LIN {X 0,Y 517.582,Z 524.387,A -85,B 0,C 180,E1 -5009.502,E2 -5009.502} C_VEL
LIN {X 0,Y 517.228,Z 535.267,A -85,B 0,C 180,E1 -5010.714,E2 -5010.714} C_VEL
LIN {X 0,Y 516.853,Z 543.976,A -85,B 0,C 180,E1 -5011.889,E2 -5011.889} C_VEL
LIN {X 0,Y 516.66,Z 551.467,A -85,B 0,C 180,E1 -5013.109,E2 -5013.109} C_VEL
LIN {X 0,Y 516.519,Z 557.024,A -85,B 0,C 180,E1 -5014.189,E2 -5014.189} C_VEL
LIN {X 0,Y 516.363,Z 563.536,A -85,B 0,C 180,E1 -5015.768,E2 -5015.768} C_VEL
LIN {X 0,Y 516.294,Z 567.941,A -85,B 0,C 180,E1 -5017.173,E2 -5017.173} C_VEL
LIN {X 0,Y 516.226,Z 570.925,A -85,B 0,C 180,E1 -5018.433,E2 -5018.433} C_VEL
LIN {X 0,Y 516.199,Z 573.444,A -85,B 0,C 180,E1 -5020.1,E2 -5020.1} C_VEL
LIN {X 0,Y 516.154,Z 574.446,A -85,B 0,C 180,E1 -5021.749,E2 -5021.749} C_VEL
LIN {X 0,Y 516.194,Z 574.398,A -85,B 0,C 180,E1 -5022.57,E2 -5022.57} C_VEL
LIN {X 0,Y 516.141,Z 573.229,A -85,B 0,C 180,E1 -5024.197,E2 -5024.197} C_VEL
LIN {X 0,Y 516.214,Z 570.618,A -85,B 0,C 180,E1 -5025.814,E2 -5025.814} C_VEL
LIN {X 0,Y 516.335,Z 566.52,A -85,B 0,C 180,E1 -5027.421,E2 -5027.421} C_VEL
LIN {X 0,Y 516.436,Z 560.9,A -85,B 0,C 180,E1 -5029.017,E2 -5029.017} C_VEL
LIN {X 0,Y 516.594,Z 554.564,A -85,B 0,C 180,E1 -5030.406,E2 -5030.406} C_VEL
LIN {X 0,Y 516.803,Z 546.711,A -85,B 0,C 180,E1 -5031.791,E2 -5031.791} C_VEL
LIN {X 0,Y 517.103,Z 538.503,A -85,B 0,C 180,E1 -5032.974,E2 -5032.974} C_VEL
LIN {X 0,Y 517.456,Z 528.649,A -85,B 0,C 180,E1 -5034.153,E2 -5034.153} C_VEL
LIN {X 0,Y 517.845,Z 517.719,A -85,B 0,C 180,E1 -5035.232,E2 -5035.232} C_VEL
LIN {X 0,Y 518.215,Z 506.878,A -85,B 0,C 180,E1 -5036.112,E2 -5036.112} C_VEL
LIN {X 0,Y 518.592,Z 495.168,A -85,B 0,C 180,E1 -5036.892,E2 -5036.892} C_VEL
LIN {X 0,Y 518.99,Z 482.323,A -85,B 0,C 180,E1 -5037.574,E2 -5037.574} C_VEL
LIN {X 0,Y 519.323,Z 468.411,A -85,B 0,C 180,E1 -5038.134,E2 -5038.134} C_VEL
LIN {X 0,Y 519.295,Z 460.742,A -85,B 0,C 180,E1 -5038.376,E2 -5038.376} C_VEL
LIN {X 0,Y 516.314,Z 447.75,A -85,B 0,C 180,E1 -5038.781,E2 -5038.781} C_VEL
LIN {X 0,Y 516.336,Z 445.185,A -85,B 0,C 180,E1 -5041.56,E2 -5041.56} C_VEL
LIN {X 0,Y 516.516,Z 443.11,A -85,B 0,C 180,E1 -5043.901,E2 -5043.901} C_VEL
LIN {X 0,Y 516.559,Z 440.324,A -85,B 0,C 180,E1 -5047.033,E2 -5047.033} C_VEL
LIN {X 0,Y 516.578,Z 438.281,A -85,B 0,C 180,E1 -5049.396,E2 -5049.396} C_VEL
LIN {X 0,Y 516.651,Z 436.223,A -85,B 0,C 180,E1 -5051.773,E2 -5051.773} C_VEL
LIN {X 0,Y 516.721,Z 433.411,A -85,B 0,C 180,E1 -5055.058,E2 -5055.058} C_VEL
LIN {X 0,Y 516.78,Z 430.702,A -85,B 0,C 180,E1 -5058.227,E2 -5058.227} C_VEL
LIN {X 0,Y 516.821,Z 429.737,A -85,B 0,C 180,E1 -5059.875,E2 -5059.875} C_VEL
LIN {X 0,Y 516.877,Z 429.729,A -85,B 0,C 180,E1 -5062.395,E2 -5062.395} C_VEL
LIN {X 0,Y 516.906,Z 429.721,A -85,B 0,C 180,E1 -5064.928,E2 -5064.928} C_VEL
LIN {X 0,Y 516.922,Z 429.723,A -85,B 0,C 180,E1 -5067.906,E2 -5067.906} C_VEL
LIN {X 0,Y 516.897,Z 429.726,A -85,B 0,C 180,E1 -5070.203,E2 -5070.203} C_VEL
LIN {X 0,Y 516.893,Z 429.722,A -85,B 0,C 180,E1 -5072.947,E2 -5072.947} C_VEL
LIN {X 0,Y 516.886,Z 429.728,A -85,B 0,C 180,E1 -5075.779,E2 -5075.779} C_VEL
LIN {X 0,Y 516.882,Z 429.724,A -85,B 0,C 180,E1 -5078.716,E2 -5078.716} C_VEL
LIN {X 0,Y 516.915,Z 429.724,A -85,B 0,C 180,E1 -5081.775,E2 -5081.775} C_VEL
LIN {X 0,Y 516.919,Z 429.724,A -85,B 0,C 180,E1 -5085.011,E2 -5085.011} C_VEL
LIN {X 0,Y 516.903,Z 429.871,A -85,B 0,C 180,E1 -5087.039,E2 -5087.039} C_VEL
LIN {X 0,Y 517.709,Z 434.112,A -85,B 0,C 180,E1 -5089.483,E2 -5089.483} C_VEL
LIN {X 0,Y 518.164,Z 437.995,A -85,B 0,C 180,E1 -5091.399,E2 -5091.399} C_VEL
LIN {X 0,Y 517.907,Z 443.605,A -85,B 0,C 180,E1 -5093.823,E2 -5093.823} C_VEL
LIN {X 0,Y 517.585,Z 450.744,A -85,B 0,C 180,E1 -5096.639,E2 -5096.639} C_VEL
LIN {X 0,Y 517.384,Z 456.944,A -85,B 0,C 180,E1 -5098.924,E2 -5098.924} C_VEL
LIN {X 0,Y 517.204,Z 465.92,A -85,B 0,C 180,E1 -5102.037,E2 -5102.037} C_VEL
LIN {X 0,Y 517.018,Z 473.813,A -85,B 0,C 180,E1 -5104.648,E2 -5104.648} C_VEL
LIN {X 0,Y 516.875,Z 483.182,A -85,B 0,C 180,E1 -5107.622,E2 -5107.622} C_VEL
LIN {X 0,Y 516.76,Z 492.685,A -85,B 0,C 180,E1 -5110.537,E2 -5110.537} C_VEL
LIN {X 0,Y 516.657,Z 501.369,A -85,B 0,C 180,E1 -5113.199,E2 -5113.199} C_VEL
LIN {X 0,Y 519.498,Z 516.364,A -85,B 0,C 180,E1 -5113.597,E2 -5113.597} C_VEL
LIN {X 0,Y 519.215,Z 529.798,A -85,B 0,C 180,E1 -5114.012,E2 -5114.012} C_VEL
LIN {X 0,Y 518.816,Z 543.3,A -85,B 0,C 180,E1 -5114.583,E2 -5114.583} C_VEL
LIN {X 0,Y 518.474,Z 555.946,A -85,B 0,C 180,E1 -5115.277,E2 -5115.277} C_VEL
LIN {X 0,Y 518.033,Z 568.91,A -85,B 0,C 180,E1 -5116.166,E2 -5116.166} C_VEL
LIN {X 0,Y 517.648,Z 580.606,A -85,B 0,C 180,E1 -5117.155,E2 -5117.155} C_VEL
LIN {X 0,Y 517.328,Z 591.208,A -85,B 0,C 180,E1 -5118.242,E2 -5118.242} C_VEL
LIN {X 0,Y 517.002,Z 600.782,A -85,B 0,C 180,E1 -5119.426,E2 -5119.426} C_VEL
LIN {X 0,Y 516.77,Z 608.636,A -85,B 0,C 180,E1 -5120.608,E2 -5120.608} C_VEL
LIN {X 0,Y 516.576,Z 615.134,A -85,B 0,C 180,E1 -5121.787,E2 -5121.787} C_VEL
LIN {X 0,Y 516.406,Z 620.528,A -85,B 0,C 180,E1 -5122.965,E2 -5122.965} C_VEL
LIN {X 0,Y 516.407,Z 624.961,A -85,B 0,C 180,E1 -5124.142,E2 -5124.142} C_VEL
LIN {X 0,Y 516.264,Z 628.444,A -85,B 0,C 180,E1 -5125.315,E2 -5125.315} C_VEL
LIN {X 0,Y 516.276,Z 631.832,A -85,B 0,C 180,E1 -5126.879,E2 -5126.879} C_VEL
LIN {X 0,Y 516.188,Z 633.835,A -85,B 0,C 180,E1 -5128.44,E2 -5128.44} C_VEL
LIN {X 0,Y 516.152,Z 634.5,A -85,B 0,C 180,E1 -5130,E2 -5130} C_VEL
LIN {X 0,Y 516.188,Z 633.837,A -85,B 0,C 180,E1 -5131.56,E2 -5131.56} C_VEL
LIN {X 0,Y 516.276,Z 631.836,A -85,B 0,C 180,E1 -5133.121,E2 -5133.121} C_VEL
LIN {X 0,Y 516.325,Z 630.32,A -85,B 0,C 180,E1 -5133.902,E2 -5133.902} C_VEL
LIN {X 0,Y 516.388,Z 626.201,A -85,B 0,C 180,E1 -5135.467,E2 -5135.467} C_VEL
LIN {X 0,Y 516.406,Z 620.526,A -85,B 0,C 180,E1 -5137.035,E2 -5137.035} C_VEL
LIN {X 0,Y 516.599,Z 614.127,A -85,B 0,C 180,E1 -5138.409,E2 -5138.409} C_VEL
LIN {X 0,Y 516.826,Z 606.174,A -85,B 0,C 180,E1 -5139.786,E2 -5139.786} C_VEL
LIN {X 0,Y 517.109,Z 597.777,A -85,B 0,C 180,E1 -5140.969,E2 -5140.969} C_VEL
LIN {X 0,Y 517.439,Z 587.23,A -85,B 0,C 180,E1 -5142.197,E2 -5142.197} C_VEL
LIN {X 0,Y 517.815,Z 576.321,A -85,B 0,C 180,E1 -5143.24,E2 -5143.24} C_VEL
LIN {X 0,Y 518.231,Z 563.637,A -85,B 0,C 180,E1 -5144.229,E2 -5144.229} C_VEL
LIN {X 0,Y 518.694,Z 551.059,A -85,B 0,C 180,E1 -5145.018,E2 -5145.018} C_VEL
LIN {X 0,Y 519.021,Z 538.132,A -85,B 0,C 180,E1 -5145.662,E2 -5145.662} C_VEL
LIN {X 0,Y 519.346,Z 524.193,A -85,B 0,C 180,E1 -5146.186,E2 -5146.186} C_VEL
LIN {X 0,Y 519.351,Z 515.338,A -85,B 0,C 180,E1 -5146.444,E2 -5146.444} C_VEL
LIN {X 0,Y 516.657,Z 501.675,A -85,B 0,C 180,E1 -5146.801,E2 -5146.801} C_VEL
LIN {X 0,Y 516.81,Z 491.833,A -85,B 0,C 180,E1 -5149.875,E2 -5149.875} C_VEL
LIN {X 0,Y 516.966,Z 482.641,A -85,B 0,C 180,E1 -5152.795,E2 -5152.795} C_VEL
LIN {X 0,Y 517.164,Z 473.559,A -85,B 0,C 180,E1 -5155.776,E2 -5155.776} C_VEL
LIN {X 0,Y 517.398,Z 464.561,A -85,B 0,C 180,E1 -5158.829,E2 -5158.829} C_VEL
LIN {X 0,Y 517.651,Z 456.874,A -85,B 0,C 180,E1 -5161.536,E2 -5161.536} C_VEL
LIN {X 0,Y 517.857,Z 449.76,A -85,B 0,C 180,E1 -5164.121,E2 -5164.121} C_VEL
LIN {X 0,Y 518.122,Z 442.579,A -85,B 0,C 180,E1 -5166.841,E2 -5166.841} C_VEL
LIN {X 0,Y 518.252,Z 438.106,A -85,B 0,C 180,E1 -5168.594,E2 -5168.594} C_VEL
LIN {X 0,Y 517.521,Z 433.141,A -85,B 0,C 180,E1 -5170.68,E2 -5170.68} C_VEL
LIN {X 0,Y 516.901,Z 429.726,A -85,B 0,C 180,E1 -5172.234,E2 -5172.234} C_VEL
LIN {X 0,Y 516.919,Z 429.724,A -85,B 0,C 180,E1 -5175.01,E2 -5175.01} C_VEL
LIN {X 0,Y 516.913,Z 429.72,A -85,B 0,C 180,E1 -5178.398,E2 -5178.398} C_VEL
LIN {X 0,Y 516.878,Z 429.726,A -85,B 0,C 180,E1 -5181.284,E2 -5181.284} C_VEL
LIN {X 0,Y 516.882,Z 429.725,A -85,B 0,C 180,E1 -5184.221,E2 -5184.221} C_VEL
LIN {X 0,Y 516.893,Z 429.725,A -85,B 0,C 180,E1 -5187.053,E2 -5187.053} C_VEL
LIN {X 0,Y 516.897,Z 429.725,A -85,B 0,C 180,E1 -5189.797,E2 -5189.797} C_VEL
LIN {X 0,Y 516.925,Z 429.72,A -85,B 0,C 180,E1 -5192.467,E2 -5192.467} C_VEL
LIN {X 0,Y 516.906,Z 429.723,A -85,B 0,C 180,E1 -5195.072,E2 -5195.072} C_VEL
LIN {X 0,Y 516.881,Z 429.729,A -85,B 0,C 180,E1 -5198.462,E2 -5198.462} C_VEL
LIN {X 0,Y 516.899,Z 429.726,A -85,B 0,C 180,E1 -5200.955,E2 -5200.955} C_VEL
LIN {X 0,Y 516.912,Z 429.722,A -85,B 0,C 180,E1 -5203.41,E2 -5203.41} C_VEL
LIN {X 0,Y 516.888,Z 429.723,A -85,B 0,C 180,E1 -5205.834,E2 -5205.834} C_VEL
LIN {X 0,Y 516.951,Z 429.718,A -85,B 0,C 180,E1 -5209.028,E2 -5209.028} C_VEL
LIN {X 0,Y 516.972,Z 429.717,A -85,B 0,C 180,E1 -5212.187,E2 -5212.187} C_VEL
LIN {X 0,Y 517.026,Z 429.708,A -85,B 0,C 180,E1 -5214.54,E2 -5214.54} C_VEL
LIN {X 0,Y 517.078,Z 429.703,A -85,B 0,C 180,E1 -5217.663,E2 -5217.663} C_VEL
LIN {X 0,Y 517.088,Z 429.7,A -85,B 0,C 180,E1 -5220.779,E2 -5220.779} C_VEL
LIN {X 0,Y 517.011,Z 429.711,A -85,B 0,C 180,E1 -5223.117,E2 -5223.117} C_VEL
LIN {X 0,Y 517.01,Z 429.71,A -85,B 0,C 180,E1 -5226.243,E2 -5226.243} C_VEL
LIN {X 0,Y 516.951,Z 429.716,A -85,B 0,C 180,E1 -5229.389,E2 -5229.389} C_VEL
LIN {X 0,Y 516.945,Z 429.718,A -85,B 0,C 180,E1 -5231.808,E2 -5231.808} C_VEL
LIN {X 0,Y 516.938,Z 429.72,A -85,B 0,C 180,E1 -5235.147,E2 -5235.147} C_VEL
LIN {X 0,Y 516.92,Z 429.724,A -85,B 0,C 180,E1 -5238.223,E2 -5238.223} C_VEL
LIN {X 0,Y 516.908,Z 429.724,A -85,B 0,C 180,E1 -5240.702,E2 -5240.702} C_VEL
LIN {X 0,Y 516.906,Z 429.724,A -85,B 0,C 180,E1 -5244.073,E2 -5244.073} C_VEL
LIN {X 0,Y 516.921,Z 429.721,A -85,B 0,C 180,E1 -5246.658,E2 -5246.658} C_VEL
LIN {X 0,Y 516.907,Z 429.724,A -85,B 0,C 180,E1 -5249.525,E2 -5249.525} C_VEL
LIN {X 0,Y 516.897,Z 429.723,A -85,B 0,C 180,E1 -5252.545,E2 -5252.545} C_VEL
LIN {X 0,Y 516.877,Z 429.725,A -85,B 0,C 180,E1 -5255.333,E2 -5255.333} C_VEL
LIN {X 0,Y 516.878,Z 429.726,A -85,B 0,C 180,E1 -5257.944,E2 -5257.944} C_VEL
LIN {X 0,Y 516.881,Z 429.724,A -85,B 0,C 180,E1 -5260.742,E2 -5260.742} C_VEL
LIN {X 0,Y 516.903,Z 429.725,A -85,B 0,C 180,E1 -5262.83,E2 -5262.83} C_VEL
LIN {X 0,Y 516.921,Z 429.719,A -85,B 0,C 180,E1 -5265.011,E2 -5265.011} C_VEL
LIN {X 0,Y 516.914,Z 429.724,A -85,B 0,C 180,E1 -5268.399,E2 -5268.399} C_VEL
LIN {X 0,Y 516.892,Z 429.724,A -85,B 0,C 180,E1 -5270.313,E2 -5270.313} C_VEL
LIN {X 0,Y 516.22,Z 429.809,A -85,B 0,C 180,E1 -5270.963,E2 -5270.963} C_VEL
LIN {X 0,Y 513.369,Z 430.165,A -85,B 0,C 180,E1 -5272.019,E2 -5272.019} C_VEL
LIN {X 0,Y 510.96,Z 430.466,A -85,B 0,C 180,E1 -5272.869,E2 -5272.869} C_VEL
LIN {X 0,Y 509.92,Z 430.594,A -85,B 0,C 180,E1 -5273.526,E2 -5273.526} C_VEL
LIN {X 0,Y 509.832,Z 430.604,A -85,B 0,C 180,E1 -5273.748,E2 -5273.748} C_VEL
LIN {X 0,Y 509.863,Z 430.602,A -85,B 0,C 180,E1 -5276.54,E2 -5276.54} C_VEL
LIN {X 0,Y 509.851,Z 430.602,A -85,B 0,C 180,E1 -5279.335,E2 -5279.335} C_VEL
LIN {X 0,Y 509.896,Z 430.599,A -85,B 0,C 180,E1 -5282.055,E2 -5282.055} C_VEL
LIN {X 0,Y 509.879,Z 430.599,A -85,B 0,C 180,E1 -5284.705,E2 -5284.705} C_VEL
LIN {X 0,Y 509.829,Z 430.605,A -85,B 0,C 180,E1 -5287.458,E2 -5287.458} C_VEL
LIN {X 0,Y 509.92,Z 430.593,A -85,B 0,C 180,E1 -5289.845,E2 -5289.845} C_VEL
LIN {X 0,Y 509.886,Z 430.599,A -85,B 0,C 180,E1 -5293.175,E2 -5293.175} C_VEL
LIN {X 0,Y 509.868,Z 430.6,A -85,B 0,C 180,E1 -5295.635,E2 -5295.635} C_VEL
LIN {X 0,Y 509.917,Z 430.595,A -85,B 0,C 180,E1 -5298.875,E2 -5298.875} C_VEL
LIN {X 0,Y 509.955,Z 430.588,A -85,B 0,C 180,E1 -5302.079,E2 -5302.079} C_VEL
LIN {X 0,Y 509.979,Z 430.586,A -85,B 0,C 180,E1 -5304.464,E2 -5304.464} C_VEL
LIN {X 0,Y 510.059,Z 430.575,A -85,B 0,C 180,E1 -5307.631,E2 -5307.631} C_VEL
LIN {X 0,Y 510.067,Z 430.574,A -85,B 0,C 180,E1 -5310.789,E2 -5310.789} C_VEL
LIN {X 0,Y 509.958,Z 430.588,A -85,B 0,C 180,E1 -5313.16,E2 -5313.16} C_VEL
LIN {X 0,Y 509.984,Z 430.586,A -85,B 0,C 180,E1 -5316.329,E2 -5316.329} C_VEL
LIN {X 0,Y 509.895,Z 430.597,A -85,B 0,C 180,E1 -5319.52,E2 -5319.52} C_VEL
LIN {X 0,Y 509.909,Z 430.596,A -85,B 0,C 180,E1 -5321.931,E2 -5321.931} C_VEL
LIN {X 0,Y 509.898,Z 430.596,A -85,B 0,C 180,E1 -5325.241,E2 -5325.241} C_VEL
LIN {X 0,Y 509.885,Z 430.596,A -85,B 0,C 180,E1 -5327.998,E2 -5327.998} C_VEL
LIN {X 0,Y 509.853,Z 430.601,A -85,B 0,C 180,E1 -5331.001,E2 -5331.001} C_VEL
LIN {X 0,Y 509.873,Z 430.6,A -85,B 0,C 180,E1 -5334.425,E2 -5334.425} C_VEL
LIN {X 0,Y 509.888,Z 430.599,A -85,B 0,C 180,E1 -5337.055,E2 -5337.055} C_VEL
LIN {X 0,Y 509.859,Z 430.602,A -85,B 0,C 180,E1 -5339.75,E2 -5339.75} C_VEL
LIN {X 0,Y 509.846,Z 430.605,A -85,B 0,C 180,E1 -5342.769,E2 -5342.769} C_VEL
LIN {X 0,Y 509.695,Z 430.624,A -85,B 0,C 180,E1 -5345.557,E2 -5345.557} C_VEL
LIN {X 0,Y 509.451,Z 430.654,A -85,B 0,C 180,E1 -5347.371,E2 -5347.371} C_VEL
LIN {X 0,Y 509.404,Z 432.343,A -85,B 0,C 180,E1 -5349.411,E2 -5349.411} C_VEL
LIN {X 0,Y 509.366,Z 435.356,A -85,B 0,C 180,E1 -5352.537,E2 -5352.537} C_VEL
LIN {X 0,Y 509.316,Z 438.013,A -85,B 0,C 180,E1 -5355.271,E2 -5355.271} C_VEL
LIN {X 0,Y 509.301,Z 440.829,A -85,B 0,C 180,E1 -5358.172,E2 -5358.172} C_VEL
LIN {X 0,Y 509.23,Z 443.23,A -85,B 0,C 180,E1 -5360.611,E2 -5360.611} C_VEL
LIN {X 0,Y 509.173,Z 446.185,A -85,B 0,C 180,E1 -5363.593,E2 -5363.593} C_VEL
LIN {X 0,Y 509.185,Z 447.643,A -85,B 0,C 180,E1 -5365.053,E2 -5365.053} C_VEL
LIN {X 0,Y 512.553,Z 462.05,A -85,B 0,C 180,E1 -5365.528,E2 -5365.528} C_VEL
LIN {X 0,Y 512.339,Z 475.814,A -85,B 0,C 180,E1 -5366.014,E2 -5366.014} C_VEL
LIN {X 0,Y 511.944,Z 488.952,A -85,B 0,C 180,E1 -5366.634,E2 -5366.634} C_VEL
LIN {X 0,Y 511.538,Z 501.39,A -85,B 0,C 180,E1 -5367.387,E2 -5367.387} C_VEL
LIN {X 0,Y 511.091,Z 513.106,A -85,B 0,C 180,E1 -5368.266,E2 -5368.266} C_VEL
LIN {X 0,Y 510.661,Z 524.126,A -85,B 0,C 180,E1 -5369.274,E2 -5369.274} C_VEL
LIN {X 0,Y 510.337,Z 533.322,A -85,B 0,C 180,E1 -5370.279,E2 -5370.279} C_VEL
LIN {X 0,Y 509.919,Z 543.164,A -85,B 0,C 180,E1 -5371.58,E2 -5371.58} C_VEL
LIN {X 0,Y 509.658,Z 551.503,A -85,B 0,C 180,E1 -5372.931,E2 -5372.931} C_VEL
LIN {X 0,Y 509.447,Z 558.111,A -85,B 0,C 180,E1 -5374.243,E2 -5374.243} C_VEL
LIN {X 0,Y 509.33,Z 563.618,A -85,B 0,C 180,E1 -5375.6,E2 -5375.6} C_VEL
LIN {X 0,Y 509.23,Z 567.618,A -85,B 0,C 180,E1 -5376.838,E2 -5376.838} C_VEL
LIN {X 0,Y 509.176,Z 570.752,A -85,B 0,C 180,E1 -5378.119,E2 -5378.119} C_VEL
LIN {X 0,Y 509.132,Z 572.341,A -85,B 0,C 180,E1 -5378.967,E2 -5378.967} C_VEL
LIN {X 0,Y 509.092,Z 574.299,A -85,B 0,C 180,E1 -5380.651,E2 -5380.651} C_VEL
LIN {X 0,Y 509.099,Z 574.776,A -85,B 0,C 180,E1 -5382.319,E2 -5382.319} C_VEL
LIN {X 0,Y 509.047,Z 573.836,A -85,B 0,C 180,E1 -5383.971,E2 -5383.971} C_VEL
LIN {X 0,Y 509.118,Z 571.48,A -85,B 0,C 180,E1 -5385.612,E2 -5385.612} C_VEL
LIN {X 0,Y 509.258,Z 567.68,A -85,B 0,C 180,E1 -5387.243,E2 -5387.243} C_VEL
LIN {X 0,Y 509.312,Z 563.858,A -85,B 0,C 180,E1 -5388.439,E2 -5388.439} C_VEL
LIN {X 0,Y 509.45,Z 558.988,A -85,B 0,C 180,E1 -5389.669,E2 -5389.669} C_VEL
LIN {X 0,Y 509.633,Z 552.069,A -85,B 0,C 180,E1 -5391.075,E2 -5391.075} C_VEL
LIN {X 0,Y 509.959,Z 543.497,A -85,B 0,C 180,E1 -5392.477,E2 -5392.477} C_VEL
LIN {X 0,Y 510.297,Z 534.568,A -85,B 0,C 180,E1 -5393.674,E2 -5393.674} C_VEL
LIN {X 0,Y 510.667,Z 523.806,A -85,B 0,C 180,E1 -5394.868,E2 -5394.868} C_VEL
LIN {X 0,Y 511.069,Z 512.891,A -85,B 0,C 180,E1 -5395.86,E2 -5395.86} C_VEL
LIN {X 0,Y 511.544,Z 500.871,A -85,B 0,C 180,E1 -5396.751,E2 -5396.751} C_VEL
LIN {X 0,Y 511.949,Z 489.396,A -85,B 0,C 180,E1 -5397.443,E2 -5397.443} C_VEL
LIN {X 0,Y 512.396,Z 475.758,A -85,B 0,C 180,E1 -5398.084,E2 -5398.084} C_VEL
LIN {X 0,Y 512.533,Z 462.151,A -85,B 0,C 180,E1 -5398.563,E2 -5398.563} C_VEL
LIN {X 0,Y 509.833,Z 450.501,A -85,B 0,C 180,E1 -5398.951,E2 -5398.951} C_VEL
LIN {X 0,Y 509.262,Z 448.284,A -85,B 0,C 180,E1 -5399.011,E2 -5399.011} C_VEL
LIN {X 0,Y 509.279,Z 445.95,A -85,B 0,C 180,E1 -5401.581,E2 -5401.581} C_VEL
LIN {X 0,Y 509.47,Z 443.813,A -85,B 0,C 180,E1 -5403.955,E2 -5403.955} C_VEL
LIN {X 0,Y 509.518,Z 441.038,A -85,B 0,C 180,E1 -5407.131,E2 -5407.131} C_VEL
LIN {X 0,Y 509.524,Z 438.956,A -85,B 0,C 180,E1 -5409.527,E2 -5409.527} C_VEL
LIN {X 0,Y 509.606,Z 436.898,A -85,B 0,C 180,E1 -5411.939,E2 -5411.939} C_VEL
LIN {X 0,Y 509.68,Z 434.149,A -85,B 0,C 180,E1 -5415.188,E2 -5415.188} C_VEL
LIN {X 0,Y 509.756,Z 431.418,A -85,B 0,C 180,E1 -5418.488,E2 -5418.488} C_VEL
LIN {X 0,Y 509.761,Z 430.758,A -85,B 0,C 180,E1 -5419.322,E2 -5419.322} C_VEL
LIN {X 0,Y 509.807,Z 430.61,A -85,B 0,C 180,E1 -5421.852,E2 -5421.852} C_VEL
LIN {X 0,Y 509.854,Z 430.603,A -85,B 0,C 180,E1 -5424.529,E2 -5424.529} C_VEL
LIN {X 0,Y 509.882,Z 430.596,A -85,B 0,C 180,E1 -5427.056,E2 -5427.056} C_VEL
LIN {X 0,Y 509.875,Z 430.599,A -85,B 0,C 180,E1 -5429.75,E2 -5429.75} C_VEL
LIN {X 0,Y 509.872,Z 430.597,A -85,B 0,C 180,E1 -5432.775,E2 -5432.775} C_VEL
LIN {X 0,Y 509.838,Z 430.604,A -85,B 0,C 180,E1 -5435.582,E2 -5435.582} C_VEL
LIN {X 0,Y 509.847,Z 430.603,A -85,B 0,C 180,E1 -5438.338,E2 -5438.338} C_VEL
LIN {X 0,Y 509.862,Z 430.601,A -85,B 0,C 180,E1 -5441.425,E2 -5441.425} C_VEL
LIN {X 0,Y 509.853,Z 430.605,A -85,B 0,C 180,E1 -5444.668,E2 -5444.668} C_VEL
LIN {X 0,Y 509.864,Z 430.81,A -85,B 0,C 180,E1 -5446.647,E2 -5446.647} C_VEL
LIN {X 0,Y 510.85,Z 436.046,A -85,B 0,C 180,E1 -5449.715,E2 -5449.715} C_VEL
LIN {X 0,Y 511.211,Z 440.221,A -85,B 0,C 180,E1 -5451.783,E2 -5451.783} C_VEL
LIN {X 0,Y 510.839,Z 447.028,A -85,B 0,C 180,E1 -5454.703,E2 -5454.703} C_VEL
LIN {X 0,Y 510.496,Z 454.238,A -85,B 0,C 180,E1 -5457.527,E2 -5457.527} C_VEL
LIN {X 0,Y 510.327,Z 460.494,A -85,B 0,C 180,E1 -5459.823,E2 -5459.823} C_VEL
LIN {X 0,Y 510.071,Z 469.506,A -85,B 0,C 180,E1 -5462.956,E2 -5462.956} C_VEL
LIN {X 0,Y 509.877,Z 478.717,A -85,B 0,C 180,E1 -5466.008,E2 -5466.008} C_VEL
LIN {X 0,Y 509.742,Z 486.765,A -85,B 0,C 180,E1 -5468.57,E2 -5468.57} C_VEL
LIN {X 0,Y 509.638,Z 496.174,A -85,B 0,C 180,E1 -5471.508,E2 -5471.508} C_VEL
LIN {X 0,Y 509.567,Z 500.902,A -85,B 0,C 180,E1 -5472.968,E2 -5472.968} C_VEL
LIN {X 0,Y 511.963,Z 513.726,A -85,B 0,C 180,E1 -5473.302,E2 -5473.302} C_VEL
LIN {X 0,Y 512.586,Z 518.364,A -85,B 0,C 180,E1 -5473.446,E2 -5473.446} C_VEL
LIN {X 0,Y 512.279,Z 532.267,A -85,B 0,C 180,E1 -5473.914,E2 -5473.914} C_VEL
LIN {X 0,Y 511.88,Z 544.613,A -85,B 0,C 180,E1 -5474.471,E2 -5474.471} C_VEL
LIN {X 0,Y 511.453,Z 558.471,A -85,B 0,C 180,E1 -5475.273,E2 -5475.273} C_VEL
LIN {X 0,Y 510.973,Z 570.86,A -85,B 0,C 180,E1 -5476.174,E2 -5476.174} C_VEL
LIN {X 0,Y 510.562,Z 582.106,A -85,B 0,C 180,E1 -5477.176,E2 -5477.176} C_VEL
LIN {X 0,Y 510.255,Z 592.36,A -85,B 0,C 180,E1 -5478.278,E2 -5478.278} C_VEL
LIN {X 0,Y 509.889,Z 601.645,A -85,B 0,C 180,E1 -5479.477,E2 -5479.477} C_VEL
LIN {X 0,Y 509.604,Z 610.518,A -85,B 0,C 180,E1 -5480.875,E2 -5480.875} C_VEL
LIN {X 0,Y 509.424,Z 616.768,A -85,B 0,C 180,E1 -5482.07,E2 -5482.07} C_VEL
LIN {X 0,Y 509.308,Z 623.403,A -85,B 0,C 180,E1 -5483.662,E2 -5483.662} C_VEL
LIN {X 0,Y 509.239,Z 627.283,A -85,B 0,C 180,E1 -5484.853,E2 -5484.853} C_VEL
LIN {X 0,Y 509.218,Z 630.271,A -85,B 0,C 180,E1 -5486.043,E2 -5486.043} C_VEL
LIN {X 0,Y 509.159,Z 632.991,A -85,B 0,C 180,E1 -5487.627,E2 -5487.627} C_VEL
LIN {X 0,Y 509.071,Z 634.33,A -85,B 0,C 180,E1 -5489.209,E2 -5489.209} C_VEL
LIN {X 0,Y 509.071,Z 634.33,A -85,B 0,C 180,E1 -5490.791,E2 -5490.791} C_VEL
LIN {X 0,Y 509.159,Z 632.994,A -85,B 0,C 180,E1 -5492.373,E2 -5492.373} C_VEL
LIN {X 0,Y 509.218,Z 630.276,A -85,B 0,C 180,E1 -5493.957,E2 -5493.957} C_VEL
LIN {X 0,Y 509.301,Z 626.092,A -85,B 0,C 180,E1 -5495.543,E2 -5495.543} C_VEL
LIN {X 0,Y 509.329,Z 620.324,A -85,B 0,C 180,E1 -5497.134,E2 -5497.134} C_VEL
LIN {X 0,Y 509.535,Z 613.831,A -85,B 0,C 180,E1 -5498.527,E2 -5498.527} C_VEL
LIN {X 0,Y 509.762,Z 605.761,A -85,B 0,C 180,E1 -5499.923,E2 -5499.923} C_VEL
LIN {X 0,Y 510.066,Z 597.324,A -85,B 0,C 180,E1 -5501.122,E2 -5501.122} C_VEL
LIN {X 0,Y 510.41,Z 587.128,A -85,B 0,C 180,E1 -5502.328,E2 -5502.328} C_VEL
LIN {X 0,Y 510.839,Z 575.836,A -85,B 0,C 180,E1 -5503.424,E2 -5503.424} C_VEL
LIN {X 0,Y 511.27,Z 563.136,A -85,B 0,C 180,E1 -5504.427,E2 -5504.427} C_VEL
LIN {X 0,Y 511.772,Z 550.544,A -85,B 0,C 180,E1 -5505.226,E2 -5505.226} C_VEL
LIN {X 0,Y 512.165,Z 537.602,A -85,B 0,C 180,E1 -5505.877,E2 -5505.877} C_VEL
LIN {X 0,Y 512.472,Z 523.802,A -85,B 0,C 180,E1 -5506.404,E2 -5506.404} C_VEL
LIN {X 0,Y 512.475,Z 516.194,A -85,B 0,C 180,E1 -5506.632,E2 -5506.632} C_VEL
LIN {X 0,Y 509.592,Z 501.309,A -85,B 0,C 180,E1 -5507.041,E2 -5507.041} C_VEL
LIN {X 0,Y 509.755,Z 491.493,A -85,B 0,C 180,E1 -5510.162,E2 -5510.162} C_VEL
LIN {X 0,Y 509.935,Z 482.371,A -85,B 0,C 180,E1 -5513.128,E2 -5513.128} C_VEL
LIN {X 0,Y 510.16,Z 473.342,A -85,B 0,C 180,E1 -5516.157,E2 -5516.157} C_VEL
LIN {X 0,Y 510.389,Z 464.396,A -85,B 0,C 180,E1 -5519.263,E2 -5519.263} C_VEL
LIN {X 0,Y 510.65,Z 456.782,A -85,B 0,C 180,E1 -5521.996,E2 -5521.996} C_VEL
LIN {X 0,Y 510.933,Z 449.238,A -85,B 0,C 180,E1 -5524.808,E2 -5524.808} C_VEL
LIN {X 0,Y 511.246,Z 441.72,A -85,B 0,C 180,E1 -5527.714,E2 -5527.714} C_VEL
LIN {X 0,Y 511.137,Z 437.999,A -85,B 0,C 180,E1 -5529.233,E2 -5529.233} C_VEL
LIN {X 0,Y 510.079,Z 431.818,A -85,B 0,C 180,E1 -5531.925,E2 -5531.925} C_VEL
LIN {X 0,Y 509.871,Z 430.601,A -85,B 0,C 180,E1 -5532.485,E2 -5532.485} C_VEL
LIN {X 0,Y 509.853,Z 430.603,A -85,B 0,C 180,E1 -5535.332,E2 -5535.332} C_VEL
LIN {X 0,Y 509.854,Z 430.6,A -85,B 0,C 180,E1 -5538.574,E2 -5538.574} C_VEL
LIN {X 0,Y 509.847,Z 430.605,A -85,B 0,C 180,E1 -5541.786,E2 -5541.786} C_VEL
LIN {X 0,Y 509.838,Z 430.605,A -85,B 0,C 180,E1 -5544.623,E2 -5544.623} C_VEL
LIN {X 0,Y 509.861,Z 430.601,A -85,B 0,C 180,E1 -5547.481,E2 -5547.481} C_VEL
LIN {X 0,Y 509.876,Z 430.6,A -85,B 0,C 180,E1 -5550.269,E2 -5550.269} C_VEL
LIN {X 0,Y 509.882,Z 430.6,A -85,B 0,C 180,E1 -5552.944,E2 -5552.944} C_VEL
LIN {X 0,Y 509.864,Z 430.602,A -85,B 0,C 180,E1 -5555.574,E2 -5555.574} C_VEL
LIN {X 0,Y 509.816,Z 430.606,A -85,B 0,C 180,E1 -5558.148,E2 -5558.148} C_VEL
LIN {X 0,Y 509.859,Z 430.601,A -85,B 0,C 180,E1 -5560.681,E2 -5560.681} C_VEL
LIN {X 0,Y 509.881,Z 430.597,A -85,B 0,C 180,E1 -5563.175,E2 -5563.175} C_VEL
LIN {X 0,Y 509.857,Z 430.6,A -85,B 0,C 180,E1 -5565.634,E2 -5565.634} C_VEL
LIN {X 0,Y 509.911,Z 430.594,A -85,B 0,C 180,E1 -5568.875,E2 -5568.875} C_VEL
LIN {X 0,Y 509.945,Z 430.591,A -85,B 0,C 180,E1 -5572.078,E2 -5572.078} C_VEL
LIN {X 0,Y 509.978,Z 430.586,A -85,B 0,C 180,E1 -5574.464,E2 -5574.464} C_VEL
LIN {X 0,Y 510.049,Z 430.578,A -85,B 0,C 180,E1 -5577.631,E2 -5577.631} C_VEL
LIN {X 0,Y 510.058,Z 430.576,A -85,B 0,C 180,E1 -5580.79,E2 -5580.79} C_VEL
LIN {X 0,Y 509.954,Z 430.59,A -85,B 0,C 180,E1 -5583.16,E2 -5583.16} C_VEL
LIN {X 0,Y 509.977,Z 430.586,A -85,B 0,C 180,E1 -5586.33,E2 -5586.33} C_VEL
LIN {X 0,Y 509.912,Z 430.595,A -85,B 0,C 180,E1 -5588.72,E2 -5588.72} C_VEL
LIN {X 0,Y 509.897,Z 430.595,A -85,B 0,C 180,E1 -5591.932,E2 -5591.932} C_VEL
LIN {X 0,Y 509.887,Z 430.598,A -85,B 0,C 180,E1 -5595.242,E2 -5595.242} C_VEL
LIN {X 0,Y 509.883,Z 430.598,A -85,B 0,C 180,E1 -5598.002,E2 -5598.002} C_VEL
LIN {X 0,Y 509.845,Z 430.604,A -85,B 0,C 180,E1 -5601.002,E2 -5601.002} C_VEL
LIN {X 0,Y 509.831,Z 430.605,A -85,B 0,C 180,E1 -5603.564,E2 -5603.564} C_VEL
LIN {X 0,Y 509.907,Z 430.597,A -85,B 0,C 180,E1 -5606.379,E2 -5606.379} C_VEL
LIN {X 0,Y 509.872,Z 430.599,A -85,B 0,C 180,E1 -5608.845,E2 -5608.845} C_VEL
LIN {X 0,Y 509.821,Z 430.604,A -85,B 0,C 180,E1 -5611.59,E2 -5611.59} C_VEL
LIN {X 0,Y 509.849,Z 430.603,A -85,B 0,C 180,E1 -5614.414,E2 -5614.414} C_VEL
LIN {X 0,Y 509.815,Z 430.607,A -85,B 0,C 180,E1 -5617.341,E2 -5617.341} C_VEL
LIN {X 0,Y 509.835,Z 430.604,A -85,B 0,C 180,E1 -5620.383,E2 -5620.383} C_VEL
LIN {X 0,Y 509.838,Z 430.604,A -85,B 0,C 180,E1 -5623.065,E2 -5623.065} C_VEL
LIN {X 0,Y 509.829,Z 430.607,A -85,B 0,C 180,E1 -5625.793,E2 -5625.793} C_VEL
LIN {X 0,Y 509.857,Z 430.602,A -85,B 0,C 180,E1 -5628.576,E2 -5628.576} C_VEL
LIN {X 0,Y 509.852,Z 430.601,A -85,B 0,C 180,E1 -5631.787,E2 -5631.787} C_VEL
LIN {X 0,Y 509.832,Z 430.604,A -85,B 0,C 180,E1 -5633.748,E2 -5633.748} C_VEL
LIN {X 0,Y 509.167,Z 430.686,A -85,B 0,C 180,E1 -5634.408,E2 -5634.408} C_VEL
LIN {X 0,Y 506.349,Z 431.04,A -85,B 0,C 180,E1 -5635.48,E2 -5635.48} C_VEL
LIN {X 0,Y 503.955,Z 431.338,A -85,B 0,C 180,E1 -5636.343,E2 -5636.343} C_VEL
LIN {X 0,Y 502.906,Z 431.467,A -85,B 0,C 180,E1 -5637.009,E2 -5637.009} C_VEL
LIN {X 0,Y 502.809,Z 431.478,A -85,B 0,C 180,E1 -5637.235,E2 -5637.235} C_VEL
LIN {X 0,Y 502.832,Z 431.476,A -85,B 0,C 180,E1 -5640.062,E2 -5640.062} C_VEL
LIN {X 0,Y 502.836,Z 431.475,A -85,B 0,C 180,E1 -5642.534,E2 -5642.534} C_VEL
LIN {X 0,Y 502.829,Z 431.477,A -85,B 0,C 180,E1 -5645.3,E2 -5645.3} C_VEL
LIN {X 0,Y 502.783,Z 431.484,A -85,B 0,C 180,E1 -5647.827,E2 -5647.827} C_VEL
LIN {X 0,Y 502.828,Z 431.478,A -85,B 0,C 180,E1 -5650.401,E2 -5650.401} C_VEL
LIN {X 0,Y 502.833,Z 431.475,A -85,B 0,C 180,E1 -5652.932,E2 -5652.932} C_VEL
LIN {X 0,Y 502.849,Z 431.474,A -85,B 0,C 180,E1 -5655.43,E2 -5655.43} C_VEL
LIN {X 0,Y 502.881,Z 431.471,A -85,B 0,C 180,E1 -5658.717,E2 -5658.717} C_VEL
LIN {X 0,Y 502.905,Z 431.466,A -85,B 0,C 180,E1 -5661.967,E2 -5661.967} C_VEL
LIN {X 0,Y 502.931,Z 431.464,A -85,B 0,C 180,E1 -5664.387,E2 -5664.387} C_VEL
LIN {X 0,Y 503.029,Z 431.451,A -85,B 0,C 180,E1 -5667.598,E2 -5667.598} C_VEL
LIN {X 0,Y 503.032,Z 431.45,A -85,B 0,C 180,E1 -5670,E2 -5670} C_VEL
LIN {X 0,Y 503.029,Z 431.452,A -85,B 0,C 180,E1 -5672.402,E2 -5672.402} C_VEL
LIN {X 0,Y 502.934,Z 431.464,A -85,B 0,C 180,E1 -5676.419,E2 -5676.419} C_VEL
LIN {X 0,Y 502.842,Z 431.474,A -85,B 0,C 180,E1 -5679.655,E2 -5679.655} C_VEL
LIN {X 0,Y 502.85,Z 431.475,A -85,B 0,C 180,E1 -5682.101,E2 -5682.101} C_VEL
LIN {X 0,Y 502.852,Z 431.473,A -85,B 0,C 180,E1 -5685.399,E2 -5685.399} C_VEL
LIN {X 0,Y 502.844,Z 431.472,A -85,B 0,C 180,E1 -5688.12,E2 -5688.12} C_VEL
LIN {X 0,Y 502.832,Z 431.478,A -85,B 0,C 180,E1 -5690.536,E2 -5690.536} C_VEL
LIN {X 0,Y 502.797,Z 431.483,A -85,B 0,C 180,E1 -5693.04,E2 -5693.04} C_VEL
LIN {X 0,Y 502.843,Z 431.476,A -85,B 0,C 180,E1 -5695.675,E2 -5695.675} C_VEL
LIN {X 0,Y 502.842,Z 431.475,A -85,B 0,C 180,E1 -5698.372,E2 -5698.372} C_VEL
LIN {X 0,Y 502.796,Z 431.48,A -85,B 0,C 180,E1 -5701.499,E2 -5701.499} C_VEL
LIN {X 0,Y 502.749,Z 431.489,A -85,B 0,C 180,E1 -5704.434,E2 -5704.434} C_VEL
LIN {X 0,Y 502.447,Z 431.527,A -85,B 0,C 180,E1 -5707.127,E2 -5707.127} C_VEL
LIN {X 0,Y 502.34,Z 431.65,A -85,B 0,C 180,E1 -5707.994,E2 -5707.994} C_VEL
LIN {X 0,Y 502.292,Z 434.638,A -85,B 0,C 180,E1 -5711.117,E2 -5711.117} C_VEL
LIN {X 0,Y 502.282,Z 437.848,A -85,B 0,C 180,E1 -5714.471,E2 -5714.471} C_VEL
LIN {X 0,Y 502.255,Z 441.138,A -85,B 0,C 180,E1 -5717.869,E2 -5717.869} C_VEL
LIN {X 0,Y 502.125,Z 444.17,A -85,B 0,C 180,E1 -5720.961,E2 -5720.961} C_VEL
LIN {X 0,Y 502.094,Z 447.156,A -85,B 0,C 180,E1 -5723.992,E2 -5723.992} C_VEL
LIN {X 0,Y 502.118,Z 448.015,A -85,B 0,C 180,E1 -5724.825,E2 -5724.825} C_VEL
LIN {X 0,Y 505.215,Z 460.703,A -85,B 0,C 180,E1 -5725.236,E2 -5725.236} C_VEL
LIN {X 0,Y 505.786,Z 464.473,A -85,B 0,C 180,E1 -5725.37,E2 -5725.37} C_VEL
LIN {X 0,Y 505.454,Z 478.554,A -85,B 0,C 180,E1 -5725.903,E2 -5725.903} C_VEL
LIN {X 0,Y 504.986,Z 492.613,A -85,B 0,C 180,E1 -5726.618,E2 -5726.618} C_VEL
LIN {X 0,Y 504.496,Z 505.331,A -85,B 0,C 180,E1 -5727.447,E2 -5727.447} C_VEL
LIN {X 0,Y 504.051,Z 516.554,A -85,B 0,C 180,E1 -5728.351,E2 -5728.351} C_VEL
LIN {X 0,Y 503.58,Z 528.202,A -85,B 0,C 180,E1 -5729.492,E2 -5729.492} C_VEL
LIN {X 0,Y 503.166,Z 538.501,A -85,B 0,C 180,E1 -5730.734,E2 -5730.734} C_VEL
LIN {X 0,Y 502.773,Z 547.627,A -85,B 0,C 180,E1 -5732.077,E2 -5732.077} C_VEL
LIN {X 0,Y 502.521,Z 555.553,A -85,B 0,C 180,E1 -5733.515,E2 -5733.515} C_VEL
LIN {X 0,Y 502.35,Z 561.067,A -85,B 0,C 180,E1 -5734.741,E2 -5734.741} C_VEL
LIN {X 0,Y 502.22,Z 565.867,A -85,B 0,C 180,E1 -5736.057,E2 -5736.057} C_VEL
LIN {X 0,Y 502.125,Z 569.864,A -85,B 0,C 180,E1 -5737.481,E2 -5737.481} C_VEL
LIN {X 0,Y 502.076,Z 572.259,A -85,B 0,C 180,E1 -5738.657,E2 -5738.657} C_VEL
LIN {X 0,Y 502.029,Z 573.838,A -85,B 0,C 180,E1 -5739.707,E2 -5739.707} C_VEL
LIN {X 0,Y 502.008,Z 575.059,A -85,B 0,C 180,E1 -5741.216,E2 -5741.216} C_VEL
LIN {X 0,Y 501.999,Z 575.053,A -85,B 0,C 180,E1 -5742.902,E2 -5742.902} C_VEL
LIN {X 0,Y 501.996,Z 573.611,A -85,B 0,C 180,E1 -5744.573,E2 -5744.573} C_VEL
LIN {X 0,Y 502.056,Z 570.751,A -85,B 0,C 180,E1 -5746.233,E2 -5746.233} C_VEL
LIN {X 0,Y 502.207,Z 566.415,A -85,B 0,C 180,E1 -5747.883,E2 -5747.883} C_VEL
LIN {X 0,Y 502.392,Z 560.5,A -85,B 0,C 180,E1 -5749.522,E2 -5749.522} C_VEL
LIN {X 0,Y 502.564,Z 553.846,A -85,B 0,C 180,E1 -5750.948,E2 -5750.948} C_VEL
LIN {X 0,Y 502.917,Z 545.547,A -85,B 0,C 180,E1 -5752.371,E2 -5752.371} C_VEL
LIN {X 0,Y 503.268,Z 536.933,A -85,B 0,C 180,E1 -5753.585,E2 -5753.585} C_VEL
LIN {X 0,Y 503.642,Z 526.544,A -85,B 0,C 180,E1 -5754.796,E2 -5754.796} C_VEL
LIN {X 0,Y 504.116,Z 514.934,A -85,B 0,C 180,E1 -5755.903,E2 -5755.903} C_VEL
LIN {X 0,Y 504.623,Z 503.296,A -85,B 0,C 180,E1 -5756.806,E2 -5756.806} C_VEL
LIN {X 0,Y 505.08,Z 490.547,A -85,B 0,C 180,E1 -5757.607,E2 -5757.607} C_VEL
LIN {X 0,Y 505.539,Z 477.235,A -85,B 0,C 180,E1 -5758.257,E2 -5758.257} C_VEL
LIN {X 0,Y 505.719,Z 463.198,A -85,B 0,C 180,E1 -5758.768,E2 -5758.768} C_VEL
LIN {X 0,Y 503.124,Z 452.274,A -85,B 0,C 180,E1 -5759.149,E2 -5759.149} C_VEL
LIN {X 0,Y 502.199,Z 448.798,A -85,B 0,C 180,E1 -5759.273,E2 -5759.273} C_VEL
LIN {X 0,Y 502.233,Z 445.969,A -85,B 0,C 180,E1 -5762.406,E2 -5762.406} C_VEL
LIN {X 0,Y 502.398,Z 443.828,A -85,B 0,C 180,E1 -5764.815,E2 -5764.815} C_VEL
LIN {X 0,Y 502.482,Z 441.75,A -85,B 0,C 180,E1 -5767.231,E2 -5767.231} C_VEL
LIN {X 0,Y 502.482,Z 439.66,A -85,B 0,C 180,E1 -5769.662,E2 -5769.662} C_VEL
LIN {X 0,Y 502.565,Z 437.599,A -85,B 0,C 180,E1 -5772.108,E2 -5772.108} C_VEL
LIN {X 0,Y 502.636,Z 434.872,A -85,B 0,C 180,E1 -5775.406,E2 -5775.406} C_VEL
LIN {X 0,Y 502.737,Z 432.173,A -85,B 0,C 180,E1 -5778.755,E2 -5778.755} C_VEL
LIN {X 0,Y 502.704,Z 431.504,A -85,B 0,C 180,E1 -5779.605,E2 -5779.605} C_VEL
LIN {X 0,Y 502.792,Z 431.482,A -85,B 0,C 180,E1 -5782.702,E2 -5782.702} C_VEL
LIN {X 0,Y 502.836,Z 431.476,A -85,B 0,C 180,E1 -5785.676,E2 -5785.676} C_VEL
LIN {X 0,Y 502.837,Z 431.477,A -85,B 0,C 180,E1 -5788.373,E2 -5788.373} C_VEL
LIN {X 0,Y 502.792,Z 431.48,A -85,B 0,C 180,E1 -5791.5,E2 -5791.5} C_VEL
LIN {X 0,Y 502.802,Z 431.48,A -85,B 0,C 180,E1 -5794.445,E2 -5794.445} C_VEL
LIN {X 0,Y 502.776,Z 431.481,A -85,B 0,C 180,E1 -5797.179,E2 -5797.179} C_VEL
LIN {X 0,Y 502.817,Z 431.48,A -85,B 0,C 180,E1 -5800.012,E2 -5800.012} C_VEL
LIN {X 0,Y 502.819,Z 431.48,A -85,B 0,C 180,E1 -5802.202,E2 -5802.202} C_VEL
LIN {X 0,Y 502.797,Z 431.485,A -85,B 0,C 180,E1 -5805.469,E2 -5805.469} C_VEL
LIN {X 0,Y 502.808,Z 431.694,A -85,B 0,C 180,E1 -5806.176,E2 -5806.176} C_VEL
LIN {X 0,Y 503.675,Z 436.265,A -85,B 0,C 180,E1 -5809.02,E2 -5809.02} C_VEL
LIN {X 0,Y 504.207,Z 440.318,A -85,B 0,C 180,E1 -5811.154,E2 -5811.154} C_VEL
LIN {X 0,Y 504.053,Z 444.731,A -85,B 0,C 180,E1 -5813.163,E2 -5813.163} C_VEL
LIN {X 0,Y 503.626,Z 451.642,A -85,B 0,C 180,E1 -5816.07,E2 -5816.07} C_VEL
LIN {X 0,Y 503.337,Z 458.977,A -85,B 0,C 180,E1 -5818.895,E2 -5818.895} C_VEL
LIN {X 0,Y 503.144,Z 466.584,A -85,B 0,C 180,E1 -5821.647,E2 -5821.647} C_VEL
LIN {X 0,Y 502.9,Z 475.69,A -85,B 0,C 180,E1 -5824.772,E2 -5824.772} C_VEL
LIN {X 0,Y 502.733,Z 484.931,A -85,B 0,C 180,E1 -5827.825,E2 -5827.825} C_VEL
LIN {X 0,Y 502.58,Z 494.302,A -85,B 0,C 180,E1 -5830.815,E2 -5830.815} C_VEL
LIN {X 0,Y 502.509,Z 500.313,A -85,B 0,C 180,E1 -5832.711,E2 -5832.711} C_VEL
LIN {X 0,Y 505.221,Z 515.394,A -85,B 0,C 180,E1 -5833.136,E2 -5833.136} C_VEL
LIN {X 0,Y 505.705,Z 518.981,A -85,B 0,C 180,E1 -5833.254,E2 -5833.254} C_VEL
LIN {X 0,Y 505.363,Z 533.326,A -85,B 0,C 180,E1 -5833.761,E2 -5833.761} C_VEL
LIN {X 0,Y 504.921,Z 545.896,A -85,B 0,C 180,E1 -5834.355,E2 -5834.355} C_VEL
LIN {X 0,Y 504.451,Z 559.322,A -85,B 0,C 180,E1 -5835.167,E2 -5835.167} C_VEL
LIN {X 0,Y 503.959,Z 571.429,A -85,B 0,C 180,E1 -5836.081,E2 -5836.081} C_VEL
LIN {X 0,Y 503.513,Z 582.499,A -85,B 0,C 180,E1 -5837.096,E2 -5837.096} C_VEL
LIN {X 0,Y 503.173,Z 593.444,A -85,B 0,C 180,E1 -5838.315,E2 -5838.315} C_VEL
LIN {X 0,Y 502.778,Z 602.478,A -85,B 0,C 180,E1 -5839.53,E2 -5839.53} C_VEL
LIN {X 0,Y 502.517,Z 611.14,A -85,B 0,C 180,E1 -5840.948,E2 -5840.948} C_VEL
LIN {X 0,Y 502.296,Z 618.119,A -85,B 0,C 180,E1 -5842.362,E2 -5842.362} C_VEL
LIN {X 0,Y 502.234,Z 622.932,A -85,B 0,C 180,E1 -5843.573,E2 -5843.573} C_VEL
LIN {X 0,Y 502.172,Z 626.831,A -85,B 0,C 180,E1 -5844.781,E2 -5844.781} C_VEL
LIN {X 0,Y 502.118,Z 629.825,A -85,B 0,C 180,E1 -5845.987,E2 -5845.987} C_VEL
LIN {X 0,Y 502.092,Z 632.575,A -85,B 0,C 180,E1 -5847.593,E2 -5847.593} C_VEL
LIN {X 0,Y 501.988,Z 633.933,A -85,B 0,C 180,E1 -5849.198,E2 -5849.198} C_VEL
LIN {X 0,Y 501.988,Z 633.938,A -85,B 0,C 180,E1 -5850.802,E2 -5850.802} C_VEL
LIN {X 0,Y 502.092,Z 632.594,A -85,B 0,C 180,E1 -5852.407,E2 -5852.407} C_VEL
LIN {X 0,Y 502.117,Z 629.862,A -85,B 0,C 180,E1 -5854.013,E2 -5854.013} C_VEL
LIN {X 0,Y 502.214,Z 625.676,A -85,B 0,C 180,E1 -5855.622,E2 -5855.622} C_VEL
LIN {X 0,Y 502.254,Z 619.901,A -85,B 0,C 180,E1 -5857.235,E2 -5857.235} C_VEL
LIN {X 0,Y 502.449,Z 613.398,A -85,B 0,C 180,E1 -5858.648,E2 -5858.648} C_VEL
LIN {X 0,Y 502.681,Z 605.318,A -85,B 0,C 180,E1 -5860.065,E2 -5860.065} C_VEL
LIN {X 0,Y 503.023,Z 596.871,A -85,B 0,C 180,E1 -5861.28,E2 -5861.28} C_VEL
LIN {X 0,Y 503.415,Z 586.049,A -85,B 0,C 180,E1 -5862.569,E2 -5862.569} C_VEL
LIN {X 0,Y 503.858,Z 575.35,A -85,B 0,C 180,E1 -5863.614,E2 -5863.614} C_VEL
LIN {X 0,Y 504.296,Z 564.075,A -85,B 0,C 180,E1 -5864.528,E2 -5864.528} C_VEL
LIN {X 0,Y 504.801,Z 551.808,A -85,B 0,C 180,E1 -5865.338,E2 -5865.338} C_VEL
LIN {X 0,Y 505.266,Z 538.209,A -85,B 0,C 180,E1 -5866.048,E2 -5866.048} C_VEL
LIN {X 0,Y 505.614,Z 523.952,A -85,B 0,C 180,E1 -5866.609,E2 -5866.609} C_VEL
LIN {X 0,Y 505.646,Z 517.254,A -85,B 0,C 180,E1 -5866.816,E2 -5866.816} C_VEL
LIN {X 0,Y 502.932,Z 503.535,A -85,B 0,C 180,E1 -5867.218,E2 -5867.218} C_VEL
LIN {X 0,Y 502.518,Z 500.942,A -85,B 0,C 180,E1 -5867.289,E2 -5867.289} C_VEL
LIN {X 0,Y 502.711,Z 491.046,A -85,B 0,C 180,E1 -5870.5,E2 -5870.5} C_VEL
LIN {X 0,Y 502.901,Z 482.123,A -85,B 0,C 180,E1 -5873.471,E2 -5873.471} C_VEL
LIN {X 0,Y 503.155,Z 472.915,A -85,B 0,C 180,E1 -5876.627,E2 -5876.627} C_VEL
LIN {X 0,Y 503.412,Z 464.35,A -85,B 0,C 180,E1 -5879.658,E2 -5879.658} C_VEL
LIN {X 0,Y 503.71,Z 456.632,A -85,B 0,C 180,E1 -5882.491,E2 -5882.491} C_VEL
LIN {X 0,Y 504.097,Z 447.836,A -85,B 0,C 180,E1 -5885.841,E2 -5885.841} C_VEL
LIN {X 0,Y 504.331,Z 441.782,A -85,B 0,C 180,E1 -5888.252,E2 -5888.252} C_VEL
LIN {X 0,Y 503.782,Z 436.639,A -85,B 0,C 180,E1 -5890.442,E2 -5890.442} C_VEL
LIN {X 0,Y 502.79,Z 431.484,A -85,B 0,C 180,E1 -5892.828,E2 -5892.828} C_VEL
LIN {X 0,Y 502.786,Z 431.482,A -85,B 0,C 180,E1 -5895.661,E2 -5895.661} C_VEL
LIN {X 0,Y 502.826,Z 431.477,A -85,B 0,C 180,E1 -5897.864,E2 -5897.864} C_VEL
LIN {X 0,Y 502.798,Z 431.48,A -85,B 0,C 180,E1 -5901.024,E2 -5901.024} C_VEL
LIN {X 0,Y 502.778,Z 431.481,A -85,B 0,C 180,E1 -5904.167,E2 -5904.167} C_VEL
LIN {X 0,Y 502.828,Z 431.477,A -85,B 0,C 180,E1 -5906.993,E2 -5906.993} C_VEL
LIN {X 0,Y 502.825,Z 431.478,A -85,B 0,C 180,E1 -5910.061,E2 -5910.061} C_VEL
LIN {X 0,Y 502.83,Z 431.476,A -85,B 0,C 180,E1 -5912.533,E2 -5912.533} C_VEL
LIN {X 0,Y 502.823,Z 431.478,A -85,B 0,C 180,E1 -5915.298,E2 -5915.298} C_VEL
LIN {X 0,Y 502.779,Z 431.481,A -85,B 0,C 180,E1 -5917.826,E2 -5917.826} C_VEL
LIN {X 0,Y 502.819,Z 431.477,A -85,B 0,C 180,E1 -5920.4,E2 -5920.4} C_VEL
LIN {X 0,Y 502.83,Z 431.476,A -85,B 0,C 180,E1 -5922.932,E2 -5922.932} C_VEL
LIN {X 0,Y 502.838,Z 431.475,A -85,B 0,C 180,E1 -5925.429,E2 -5925.429} C_VEL
LIN {X 0,Y 502.875,Z 431.47,A -85,B 0,C 180,E1 -5928.717,E2 -5928.717} C_VEL
LIN {X 0,Y 502.896,Z 431.468,A -85,B 0,C 180,E1 -5931.967,E2 -5931.967} C_VEL
LIN {X 0,Y 502.933,Z 431.463,A -85,B 0,C 180,E1 -5934.387,E2 -5934.387} C_VEL
LIN {X 0,Y 503.019,Z 431.454,A -85,B 0,C 180,E1 -5937.598,E2 -5937.598} C_VEL
LIN {X 0,Y 503.02,Z 431.451,A -85,B 0,C 180,E1 -5940,E2 -5940} C_VEL
LIN {X 0,Y 503.02,Z 431.452,A -85,B 0,C 180,E1 -5942.402,E2 -5942.402} C_VEL
LIN {X 0,Y 502.957,Z 431.461,A -85,B 0,C 180,E1 -5945.613,E2 -5945.613} C_VEL
LIN {X 0,Y 502.896,Z 431.467,A -85,B 0,C 180,E1 -5948.034,E2 -5948.034} C_VEL
LIN {X 0,Y 502.871,Z 431.472,A -85,B 0,C 180,E1 -5951.284,E2 -5951.284} C_VEL
LIN {X 0,Y 502.839,Z 431.475,A -85,B 0,C 180,E1 -5954.571,E2 -5954.571} C_VEL
LIN {X 0,Y 502.856,Z 431.473,A -85,B 0,C 180,E1 -5957.907,E2 -5957.907} C_VEL
LIN {X 0,Y 502.823,Z 431.478,A -85,B 0,C 180,E1 -5960.537,E2 -5960.537} C_VEL
LIN {X 0,Y 502.791,Z 431.48,A -85,B 0,C 180,E1 -5963.041,E2 -5963.041} C_VEL
LIN {X 0,Y 502.835,Z 431.475,A -85,B 0,C 180,E1 -5965.676,E2 -5965.676} C_VEL
LIN {X 0,Y 502.836,Z 431.475,A -85,B 0,C 180,E1 -5968.373,E2 -5968.373} C_VEL
LIN {X 0,Y 502.792,Z 431.479,A -85,B 0,C 180,E1 -5971.5,E2 -5971.5} C_VEL
LIN {X 0,Y 502.801,Z 431.481,A -85,B 0,C 180,E1 -5974.445,E2 -5974.445} C_VEL
LIN {X 0,Y 502.777,Z 431.483,A -85,B 0,C 180,E1 -5977.179,E2 -5977.179} C_VEL
LIN {X 0,Y 502.785,Z 431.483,A -85,B 0,C 180,E1 -5980.016,E2 -5980.016} C_VEL
LIN {X 0,Y 502.8,Z 431.48,A -85,B 0,C 180,E1 -5982.2,E2 -5982.2} C_VEL
LIN {X 0,Y 502.799,Z 431.48,A -85,B 0,C 180,E1 -5985.469,E2 -5985.469} C_VEL
LIN {X 0,Y 502.822,Z 431.476,A -85,B 0,C 180,E1 -5988.935,E2 -5988.935} C_VEL
LIN {X 0,Y 502.794,Z 431.481,A -85,B 0,C 180,E1 -5992.047,E2 -5992.047} C_VEL
LIN {X 0,Y 502.81,Z 431.478,A -85,B 0,C 180,E1 -5995.036,E2 -5995.036} C_VEL
LIN {X 0,Y 502.809,Z 431.478,A -85,B 0,C 180,E1 -5997.235,E2 -5997.235} C_VEL
LIN {X 0,Y 502.11,Z 431.568,A -85,B 0,C 180,E1 -5997.904,E2 -5997.904} C_VEL
LIN {X 0,Y 499.252,Z 431.92,A -85,B 0,C 180,E1 -5998.989,E2 -5998.989} C_VEL
LIN {X 0,Y 496.862,Z 432.22,A -85,B 0,C 180,E1 -5999.864,E2 -5999.864} C_VEL
LIN {X 0,Y 495.844,Z 432.348,A -85,B 0,C 180,E1 -6000.54,E2 -6000.54} C_VEL
LIN {X 0,Y 495.765,Z 432.354,A -85,B 0,C 180,E1 -6000.769,E2 -6000.769} C_VEL
LIN {X 0,Y 495.793,Z 432.353,A -85,B 0,C 180,E1 -6003.933,E2 -6003.933} C_VEL
LIN {X 0,Y 495.763,Z 432.355,A -85,B 0,C 180,E1 -6007.14,E2 -6007.14} C_VEL
LIN {X 0,Y 495.774,Z 432.356,A -85,B 0,C 180,E1 -6010.11,E2 -6010.11} C_VEL
LIN {X 0,Y 495.785,Z 432.352,A -85,B 0,C 180,E1 -6012.682,E2 -6012.682} C_VEL
LIN {X 0,Y 495.794,Z 432.352,A -85,B 0,C 180,E1 -6015.218,E2 -6015.218} C_VEL
LIN {X 0,Y 495.856,Z 432.346,A -85,B 0,C 180,E1 -6018.555,E2 -6018.555} C_VEL
LIN {X 0,Y 495.876,Z 432.342,A -85,B 0,C 180,E1 -6021.852,E2 -6021.852} C_VEL
LIN {X 0,Y 495.842,Z 432.346,A -85,B 0,C 180,E1 -6025.122,E2 -6025.122} C_VEL
LIN {X 0,Y 495.998,Z 432.327,A -85,B 0,C 180,E1 -6027.564,E2 -6027.564} C_VEL
LIN {X 0,Y 495.987,Z 432.328,A -85,B 0,C 180,E1 -6030.812,E2 -6030.812} C_VEL
LIN {X 0,Y 495.998,Z 432.328,A -85,B 0,C 180,E1 -6032.436,E2 -6032.436} C_VEL
LIN {X 0,Y 495.901,Z 432.339,A -85,B 0,C 180,E1 -6035.693,E2 -6035.693} C_VEL
LIN {X 0,Y 495.841,Z 432.347,A -85,B 0,C 180,E1 -6038.148,E2 -6038.148} C_VEL
LIN {X 0,Y 495.856,Z 432.345,A -85,B 0,C 180,E1 -6041.445,E2 -6041.445} C_VEL
LIN {X 0,Y 495.794,Z 432.354,A -85,B 0,C 180,E1 -6044.782,E2 -6044.782} C_VEL
LIN {X 0,Y 495.784,Z 432.356,A -85,B 0,C 180,E1 -6047.318,E2 -6047.318} C_VEL
LIN {X 0,Y 495.774,Z 432.355,A -85,B 0,C 180,E1 -6049.89,E2 -6049.89} C_VEL
LIN {X 0,Y 495.764,Z 432.357,A -85,B 0,C 180,E1 -6052.861,E2 -6052.861} C_VEL
LIN {X 0,Y 495.793,Z 432.353,A -85,B 0,C 180,E1 -6056.067,E2 -6056.067} C_VEL
LIN {X 0,Y 495.774,Z 432.356,A -85,B 0,C 180,E1 -6058.814,E2 -6058.814} C_VEL
LIN {X 0,Y 495.758,Z 432.355,A -85,B 0,C 180,E1 -6061.725,E2 -6061.725} C_VEL
LIN {X 0,Y 495.676,Z 432.37,A -85,B 0,C 180,E1 -6064.678,E2 -6064.678} C_VEL
LIN {X 0,Y 495.336,Z 432.412,A -85,B 0,C 180,E1 -6067.596,E2 -6067.596} C_VEL
LIN {X 0,Y 495.266,Z 432.972,A -85,B 0,C 180,E1 -6068.696,E2 -6068.696} C_VEL
LIN {X 0,Y 495.224,Z 435.956,A -85,B 0,C 180,E1 -6071.835,E2 -6071.835} C_VEL
LIN {X 0,Y 495.186,Z 438.788,A -85,B 0,C 180,E1 -6074.795,E2 -6074.795} C_VEL
LIN {X 0,Y 495.162,Z 442.03,A -85,B 0,C 180,E1 -6078.157,E2 -6078.157} C_VEL
LIN {X 0,Y 495.042,Z 445.154,A -85,B 0,C 180,E1 -6081.343,E2 -6081.343} C_VEL
LIN {X 0,Y 495.05,Z 448.323,A -85,B 0,C 180,E1 -6084.563,E2 -6084.563} C_VEL
LIN {X 0,Y 498.416,Z 461.888,A -85,B 0,C 180,E1 -6085.032,E2 -6085.032} C_VEL
LIN {X 0,Y 498.968,Z 465.945,A -85,B 0,C 180,E1 -6085.18,E2 -6085.18} C_VEL
LIN {X 0,Y 498.6,Z 479.919,A -85,B 0,C 180,E1 -6085.729,E2 -6085.729} C_VEL
LIN {X 0,Y 498.125,Z 493.461,A -85,B 0,C 180,E1 -6086.438,E2 -6086.438} C_VEL
LIN {X 0,Y 497.592,Z 506.37,A -85,B 0,C 180,E1 -6087.299,E2 -6087.299} C_VEL
LIN {X 0,Y 497.088,Z 518.509,A -85,B 0,C 180,E1 -6088.308,E2 -6088.308} C_VEL
LIN {X 0,Y 496.623,Z 529.009,A -85,B 0,C 180,E1 -6089.372,E2 -6089.372} C_VEL
LIN {X 0,Y 496.217,Z 538.402,A -85,B 0,C 180,E1 -6090.516,E2 -6090.516} C_VEL
LIN {X 0,Y 495.803,Z 547.138,A -85,B 0,C 180,E1 -6091.798,E2 -6091.798} C_VEL
LIN {X 0,Y 495.582,Z 554.02,A -85,B 0,C 180,E1 -6093.012,E2 -6093.012} C_VEL
LIN {X 0,Y 495.336,Z 560.304,A -85,B 0,C 180,E1 -6094.358,E2 -6094.358} C_VEL
LIN {X 0,Y 495.198,Z 565.324,A -85,B 0,C 180,E1 -6095.696,E2 -6095.696} C_VEL
LIN {X 0,Y 495.055,Z 570.05,A -85,B 0,C 180,E1 -6097.331,E2 -6097.331} C_VEL
LIN {X 0,Y 494.995,Z 572.178,A -85,B 0,C 180,E1 -6098.336,E2 -6098.336} C_VEL
LIN {X 0,Y 494.92,Z 574.642,A -85,B 0,C 180,E1 -6100.074,E2 -6100.074} C_VEL
LIN {X 0,Y 494.934,Z 575.609,A -85,B 0,C 180,E1 -6101.796,E2 -6101.796} C_VEL
LIN {X 0,Y 494.907,Z 575.137,A -85,B 0,C 180,E1 -6103.5,E2 -6103.5} C_VEL
LIN {X 0,Y 494.962,Z 573.234,A -85,B 0,C 180,E1 -6105.192,E2 -6105.192} C_VEL
LIN {X 0,Y 495.052,Z 569.857,A -85,B 0,C 180,E1 -6106.871,E2 -6106.871} C_VEL
LIN {X 0,Y 495.202,Z 564.968,A -85,B 0,C 180,E1 -6108.539,E2 -6108.539} C_VEL
LIN {X 0,Y 495.383,Z 560.239,A -85,B 0,C 180,E1 -6109.785,E2 -6109.785} C_VEL
LIN {X 0,Y 495.592,Z 553.403,A -85,B 0,C 180,E1 -6111.231,E2 -6111.231} C_VEL
LIN {X 0,Y 495.971,Z 544.744,A -85,B 0,C 180,E1 -6112.7,E2 -6112.7} C_VEL
LIN {X 0,Y 496.336,Z 536.098,A -85,B 0,C 180,E1 -6113.904,E2 -6113.904} C_VEL
LIN {X 0,Y 496.763,Z 525.456,A -85,B 0,C 180,E1 -6115.13,E2 -6115.13} C_VEL
LIN {X 0,Y 497.25,Z 514.681,A -85,B 0,C 180,E1 -6116.15,E2 -6116.15} C_VEL
LIN {X 0,Y 497.783,Z 502.904,A -85,B 0,C 180,E1 -6117.066,E2 -6117.066} C_VEL
LIN {X 0,Y 498.301,Z 489.883,A -85,B 0,C 180,E1 -6117.878,E2 -6117.878} C_VEL
LIN {X 0,Y 498.74,Z 477.438,A -85,B 0,C 180,E1 -6118.486,E2 -6118.486} C_VEL
LIN {X 0,Y 498.946,Z 464.633,A -85,B 0,C 180,E1 -6118.966,E2 -6118.966} C_VEL
LIN {X 0,Y 496.728,Z 454.957,A -85,B 0,C 180,E1 -6119.316,E2 -6119.316} C_VEL
LIN {X 0,Y 495.155,Z 449.322,A -85,B 0,C 180,E1 -6119.517,E2 -6119.517} C_VEL
LIN {X 0,Y 495.175,Z 446.702,A -85,B 0,C 180,E1 -6122.44,E2 -6122.44} C_VEL
LIN {X 0,Y 495.351,Z 444.565,A -85,B 0,C 180,E1 -6124.883,E2 -6124.883} C_VEL
LIN {X 0,Y 495.421,Z 442.447,A -85,B 0,C 180,E1 -6127.335,E2 -6127.335} C_VEL
LIN {X 0,Y 495.475,Z 439.685,A -85,B 0,C 180,E1 -6130.626,E2 -6130.626} C_VEL
LIN {X 0,Y 495.51,Z 437.64,A -85,B 0,C 180,E1 -6133.117,E2 -6133.117} C_VEL
LIN {X 0,Y 495.577,Z 435.6,A -85,B 0,C 180,E1 -6135.631,E2 -6135.631} C_VEL
LIN {X 0,Y 495.713,Z 433.557,A -85,B 0,C 180,E1 -6138.217,E2 -6138.217} C_VEL
LIN {X 0,Y 495.661,Z 432.372,A -85,B 0,C 180,E1 -6139.895,E2 -6139.895} C_VEL
LIN {X 0,Y 495.752,Z 432.358,A -85,B 0,C 180,E1 -6142.861,E2 -6142.861} C_VEL
LIN {X 0,Y 495.794,Z 432.356,A -85,B 0,C 180,E1 -6146.068,E2 -6146.068} C_VEL
LIN {X 0,Y 495.775,Z 432.354,A -85,B 0,C 180,E1 -6148.815,E2 -6148.815} C_VEL
LIN {X 0,Y 495.754,Z 432.359,A -85,B 0,C 180,E1 -6151.727,E2 -6151.727} C_VEL
LIN {X 0,Y 495.772,Z 432.354,A -85,B 0,C 180,E1 -6154.696,E2 -6154.696} C_VEL
LIN {X 0,Y 495.727,Z 432.362,A -85,B 0,C 180,E1 -6157.562,E2 -6157.562} C_VEL
LIN {X 0,Y 495.776,Z 432.354,A -85,B 0,C 180,E1 -6160.699,E2 -6160.699} C_VEL
LIN {X 0,Y 495.731,Z 432.365,A -85,B 0,C 180,E1 -6163.696,E2 -6163.696} C_VEL
LIN {X 0,Y 495.768,Z 432.417,A -85,B 0,C 180,E1 -6165.578,E2 -6165.578} C_VEL
LIN {X 0,Y 496.588,Z 437.029,A -85,B 0,C 180,E1 -6168.598,E2 -6168.598} C_VEL
LIN {X 0,Y 497.252,Z 441.474,A -85,B 0,C 180,E1 -6171.019,E2 -6171.019} C_VEL
LIN {X 0,Y 497.069,Z 445.78,A -85,B 0,C 180,E1 -6173.066,E2 -6173.066} C_VEL
LIN {X 0,Y 496.644,Z 452.729,A -85,B 0,C 180,E1 -6176.017,E2 -6176.017} C_VEL
LIN {X 0,Y 496.313,Z 459.987,A -85,B 0,C 180,E1 -6178.879,E2 -6178.879} C_VEL
LIN {X 0,Y 496.106,Z 466.914,A -85,B 0,C 180,E1 -6181.439,E2 -6181.439} C_VEL
LIN {X 0,Y 495.88,Z 475.312,A -85,B 0,C 180,E1 -6184.389,E2 -6184.389} C_VEL
LIN {X 0,Y 495.67,Z 484.483,A -85,B 0,C 180,E1 -6187.492,E2 -6187.492} C_VEL
LIN {X 0,Y 495.495,Z 493.776,A -85,B 0,C 180,E1 -6190.53,E2 -6190.53} C_VEL
LIN {X 0,Y 495.413,Z 499.97,A -85,B 0,C 180,E1 -6192.477,E2 -6192.477} C_VEL
LIN {X 0,Y 497.97,Z 514.25,A -85,B 0,C 180,E1 -6192.873,E2 -6192.873} C_VEL
LIN {X 0,Y 498.845,Z 519.502,A -85,B 0,C 180,E1 -6193.055,E2 -6193.055} C_VEL
LIN {X 0,Y 498.463,Z 533.672,A -85,B 0,C 180,E1 -6193.575,E2 -6193.575} C_VEL
LIN {X 0,Y 497.963,Z 547.06,A -85,B 0,C 180,E1 -6194.236,E2 -6194.236} C_VEL
LIN {X 0,Y 497.462,Z 560.112,A -85,B 0,C 180,E1 -6195.059,E2 -6195.059} C_VEL
LIN {X 0,Y 496.946,Z 571.995,A -85,B 0,C 180,E1 -6195.985,E2 -6195.985} C_VEL
LIN {X 0,Y 496.445,Z 583.888,A -85,B 0,C 180,E1 -6197.117,E2 -6197.117} C_VEL
LIN {X 0,Y 496.074,Z 594.697,A -85,B 0,C 180,E1 -6198.373,E2 -6198.373} C_VEL
LIN {X 0,Y 495.688,Z 603.326,A -85,B 0,C 180,E1 -6199.585,E2 -6199.585} C_VEL
LIN {X 0,Y 495.404,Z 611.753,A -85,B 0,C 180,E1 -6201.022,E2 -6201.022} C_VEL
LIN {X 0,Y 495.213,Z 617.632,A -85,B 0,C 180,E1 -6202.252,E2 -6202.252} C_VEL
LIN {X 0,Y 495.12,Z 623.472,A -85,B 0,C 180,E1 -6203.763,E2 -6203.763} C_VEL
LIN {X 0,Y 495.031,Z 627.459,A -85,B 0,C 180,E1 -6205.114,E2 -6205.114} C_VEL
LIN {X 0,Y 495.033,Z 630.944,A -85,B 0,C 180,E1 -6206.745,E2 -6206.745} C_VEL
LIN {X 0,Y 494.958,Z 633.003,A -85,B 0,C 180,E1 -6208.373,E2 -6208.373} C_VEL
LIN {X 0,Y 494.896,Z 633.69,A -85,B 0,C 180,E1 -6210,E2 -6210} C_VEL
LIN {X 0,Y 494.958,Z 633.026,A -85,B 0,C 180,E1 -6211.627,E2 -6211.627} C_VEL
LIN {X 0,Y 495.033,Z 630.994,A -85,B 0,C 180,E1 -6213.255,E2 -6213.255} C_VEL
LIN {X 0,Y 495.031,Z 627.542,A -85,B 0,C 180,E1 -6214.886,E2 -6214.886} C_VEL
LIN {X 0,Y 495.118,Z 623.578,A -85,B 0,C 180,E1 -6216.237,E2 -6216.237} C_VEL
LIN {X 0,Y 495.213,Z 617.779,A -85,B 0,C 180,E1 -6217.748,E2 -6217.748} C_VEL
LIN {X 0,Y 495.454,Z 610.833,A -85,B 0,C 180,E1 -6219.182,E2 -6219.182} C_VEL
LIN {X 0,Y 495.749,Z 602.21,A -85,B 0,C 180,E1 -6220.62,E2 -6220.62} C_VEL
LIN {X 0,Y 496.164,Z 592.484,A -85,B 0,C 180,E1 -6221.944,E2 -6221.944} C_VEL
LIN {X 0,Y 496.559,Z 582.329,A -85,B 0,C 180,E1 -6223.088,E2 -6223.088} C_VEL
LIN {X 0,Y 497.021,Z 571.319,A -85,B 0,C 180,E1 -6224.118,E2 -6224.118} C_VEL
LIN {X 0,Y 497.569,Z 559.288,A -85,B 0,C 180,E1 -6225.043,E2 -6225.043} C_VEL
LIN {X 0,Y 498.083,Z 545.933,A -85,B 0,C 180,E1 -6225.865,E2 -6225.865} C_VEL
LIN {X 0,Y 498.568,Z 532.753,A -85,B 0,C 180,E1 -6226.494,E2 -6226.494} C_VEL
LIN {X 0,Y 498.85,Z 518.57,A -85,B 0,C 180,E1 -6226.998,E2 -6226.998} C_VEL
LIN {X 0,Y 496.033,Z 504.092,A -85,B 0,C 180,E1 -6227.445,E2 -6227.445} C_VEL
LIN {X 0,Y 495.444,Z 500.582,A -85,B 0,C 180,E1 -6227.544,E2 -6227.544} C_VEL
LIN {X 0,Y 495.656,Z 491.242,A -85,B 0,C 180,E1 -6230.638,E2 -6230.638} C_VEL
LIN {X 0,Y 495.873,Z 481.875,A -85,B 0,C 180,E1 -6233.824,E2 -6233.824} C_VEL
LIN {X 0,Y 496.136,Z 473.304,A -85,B 0,C 180,E1 -6236.82,E2 -6236.82} C_VEL
LIN {X 0,Y 496.386,Z 465.284,A -85,B 0,C 180,E1 -6239.705,E2 -6239.705} C_VEL
LIN {X 0,Y 496.713,Z 457.715,A -85,B 0,C 180,E1 -6242.524,E2 -6242.524} C_VEL
LIN {X 0,Y 497.125,Z 449.08,A -85,B 0,C 180,E1 -6245.869,E2 -6245.869} C_VEL
LIN {X 0,Y 497.356,Z 442.697,A -85,B 0,C 180,E1 -6248.443,E2 -6248.443} C_VEL
LIN {X 0,Y 496.782,Z 437.736,A -85,B 0,C 180,E1 -6250.598,E2 -6250.598} C_VEL
LIN {X 0,Y 495.731,Z 432.362,A -85,B 0,C 180,E1 -6253.159,E2 -6253.159} C_VEL
LIN {X 0,Y 495.733,Z 432.361,A -85,B 0,C 180,E1 -6255.999,E2 -6255.999} C_VEL
LIN {X 0,Y 495.759,Z 432.356,A -85,B 0,C 180,E1 -6258.705,E2 -6258.705} C_VEL
LIN {X 0,Y 495.746,Z 432.359,A -85,B 0,C 180,E1 -6261.408,E2 -6261.408} C_VEL
LIN {X 0,Y 495.75,Z 432.358,A -85,B 0,C 180,E1 -6264.463,E2 -6264.463} C_VEL
LIN {X 0,Y 495.764,Z 432.358,A -85,B 0,C 180,E1 -6267.405,E2 -6267.405} C_VEL
LIN {X 0,Y 495.776,Z 432.356,A -85,B 0,C 180,E1 -6270.254,E2 -6270.254} C_VEL
LIN {X 0,Y 495.828,Z 432.348,A -85,B 0,C 180,E1 -6273.248,E2 -6273.248} C_VEL
LIN {X 0,Y 495.746,Z 432.359,A -85,B 0,C 180,E1 -6275.725,E2 -6275.725} C_VEL
LIN {X 0,Y 495.738,Z 432.361,A -85,B 0,C 180,E1 -6278.371,E2 -6278.371} C_VEL
LIN {X 0,Y 495.779,Z 432.357,A -85,B 0,C 180,E1 -6280.971,E2 -6280.971} C_VEL
LIN {X 0,Y 495.775,Z 432.356,A -85,B 0,C 180,E1 -6283.53,E2 -6283.53} C_VEL
LIN {X 0,Y 495.787,Z 432.352,A -85,B 0,C 180,E1 -6286.056,E2 -6286.056} C_VEL
LIN {X 0,Y 495.848,Z 432.346,A -85,B 0,C 180,E1 -6288.555,E2 -6288.555} C_VEL
LIN {X 0,Y 495.867,Z 432.343,A -85,B 0,C 180,E1 -6291.852,E2 -6291.852} C_VEL
LIN {X 0,Y 495.891,Z 432.34,A -85,B 0,C 180,E1 -6294.307,E2 -6294.307} C_VEL
LIN {X 0,Y 495.988,Z 432.329,A -85,B 0,C 180,E1 -6297.564,E2 -6297.564} C_VEL
LIN {X 0,Y 495.991,Z 432.327,A -85,B 0,C 180,E1 -6300,E2 -6300} C_VEL
LIN {X 0,Y 495.989,Z 432.328,A -85,B 0,C 180,E1 -6302.436,E2 -6302.436} C_VEL
LIN {X 0,Y 495.911,Z 432.338,A -85,B 0,C 180,E1 -6305.693,E2 -6305.693} C_VEL
LIN {X 0,Y 495.867,Z 432.343,A -85,B 0,C 180,E1 -6308.148,E2 -6308.148} C_VEL
LIN {X 0,Y 495.845,Z 432.347,A -85,B 0,C 180,E1 -6311.446,E2 -6311.446} C_VEL
LIN {X 0,Y 495.784,Z 432.353,A -85,B 0,C 180,E1 -6314.783,E2 -6314.783} C_VEL
LIN {X 0,Y 495.782,Z 432.353,A -85,B 0,C 180,E1 -6317.319,E2 -6317.319} C_VEL
LIN {X 0,Y 495.773,Z 432.357,A -85,B 0,C 180,E1 -6319.891,E2 -6319.891} C_VEL
LIN {X 0,Y 495.76,Z 432.356,A -85,B 0,C 180,E1 -6322.863,E2 -6322.863} C_VEL
LIN {X 0,Y 495.786,Z 432.354,A -85,B 0,C 180,E1 -6326.068,E2 -6326.068} C_VEL
LIN {X 0,Y 495.767,Z 432.356,A -85,B 0,C 180,E1 -6328.815,E2 -6328.815} C_VEL
LIN {X 0,Y 495.755,Z 432.357,A -85,B 0,C 180,E1 -6331.727,E2 -6331.727} C_VEL
LIN {X 0,Y 495.771,Z 432.357,A -85,B 0,C 180,E1 -6334.696,E2 -6334.696} C_VEL
LIN {X 0,Y 495.728,Z 432.363,A -85,B 0,C 180,E1 -6337.562,E2 -6337.562} C_VEL
LIN {X 0,Y 495.764,Z 432.355,A -85,B 0,C 180,E1 -6340.701,E2 -6340.701} C_VEL
LIN {X 0,Y 495.733,Z 432.36,A -85,B 0,C 180,E1 -6343.696,E2 -6343.696} C_VEL
LIN {X 0,Y 495.727,Z 432.361,A -85,B 0,C 180,E1 -6346.306,E2 -6346.306} C_VEL
LIN {X 0,Y 495.775,Z 432.354,A -85,B 0,C 180,E1 -6349.302,E2 -6349.302} C_VEL
LIN {X 0,Y 495.732,Z 432.362,A -85,B 0,C 180,E1 -6352.439,E2 -6352.439} C_VEL
LIN {X 0,Y 495.786,Z 432.356,A -85,B 0,C 180,E1 -6355.458,E2 -6355.458} C_VEL
LIN {X 0,Y 495.758,Z 432.356,A -85,B 0,C 180,E1 -6358.365,E2 -6358.365} C_VEL
LIN {X 0,Y 495.765,Z 432.354,A -85,B 0,C 180,E1 -6360.769,E2 -6360.769} C_VEL
LIN {X 0,Y 495.104,Z 432.439,A -85,B 0,C 180,E1 -6361.448,E2 -6361.448} C_VEL
LIN {X 0,Y 492.243,Z 432.794,A -85,B 0,C 180,E1 -6362.55,E2 -6362.55} C_VEL
LIN {X 0,Y 489.833,Z 433.096,A -85,B 0,C 180,E1 -6363.439,E2 -6363.439} C_VEL
LIN {X 0,Y 488.817,Z 433.221,A -85,B 0,C 180,E1 -6364.125,E2 -6364.125} C_VEL
LIN {X 0,Y 488.745,Z 433.23,A -85,B 0,C 180,E1 -6364.357,E2 -6364.357} C_VEL
LIN {X 0,Y 488.725,Z 433.232,A -85,B 0,C 180,E1 -6367.154,E2 -6367.154} C_VEL
LIN {X 0,Y 488.728,Z 433.233,A -85,B 0,C 180,E1 -6369.811,E2 -6369.811} C_VEL
LIN {X 0,Y 488.733,Z 433.23,A -85,B 0,C 180,E1 -6372.424,E2 -6372.424} C_VEL
LIN {X 0,Y 488.766,Z 433.228,A -85,B 0,C 180,E1 -6375,E2 -6375} C_VEL
LIN {X 0,Y 488.81,Z 433.223,A -85,B 0,C 180,E1 -6378.388,E2 -6378.388} C_VEL
LIN {X 0,Y 488.821,Z 433.222,A -85,B 0,C 180,E1 -6381.734,E2 -6381.734} C_VEL
LIN {X 0,Y 488.811,Z 433.222,A -85,B 0,C 180,E1 -6385.051,E2 -6385.051} C_VEL
LIN {X 0,Y 488.965,Z 433.203,A -85,B 0,C 180,E1 -6387.529,E2 -6387.529} C_VEL
LIN {X 0,Y 488.938,Z 433.206,A -85,B 0,C 180,E1 -6390.824,E2 -6390.824} C_VEL
LIN {X 0,Y 488.965,Z 433.204,A -85,B 0,C 180,E1 -6392.471,E2 -6392.471} C_VEL
LIN {X 0,Y 488.86,Z 433.216,A -85,B 0,C 180,E1 -6395.776,E2 -6395.776} C_VEL
LIN {X 0,Y 488.791,Z 433.225,A -85,B 0,C 180,E1 -6398.267,E2 -6398.267} C_VEL
LIN {X 0,Y 488.81,Z 433.223,A -85,B 0,C 180,E1 -6401.612,E2 -6401.612} C_VEL
LIN {X 0,Y 488.766,Z 433.23,A -85,B 0,C 180,E1 -6405,E2 -6405} C_VEL
LIN {X 0,Y 488.758,Z 433.227,A -85,B 0,C 180,E1 -6408.442,E2 -6408.442} C_VEL
LIN {X 0,Y 488.71,Z 433.235,A -85,B 0,C 180,E1 -6411.07,E2 -6411.07} C_VEL
LIN {X 0,Y 488.696,Z 433.236,A -85,B 0,C 180,E1 -6413.745,E2 -6413.745} C_VEL
LIN {X 0,Y 488.794,Z 433.226,A -85,B 0,C 180,E1 -6416.943,E2 -6416.943} C_VEL
LIN {X 0,Y 488.711,Z 433.235,A -85,B 0,C 180,E1 -6420.362,E2 -6420.362} C_VEL
LIN {X 0,Y 488.702,Z 433.236,A -85,B 0,C 180,E1 -6423.478,E2 -6423.478} C_VEL
LIN {X 0,Y 488.46,Z 433.269,A -85,B 0,C 180,E1 -6426.318,E2 -6426.318} C_VEL
LIN {X 0,Y 488.219,Z 433.299,A -85,B 0,C 180,E1 -6428.242,E2 -6428.242} C_VEL
LIN {X 0,Y 488.154,Z 436.29,A -85,B 0,C 180,E1 -6431.526,E2 -6431.526} C_VEL
LIN {X 0,Y 488.11,Z 439.489,A -85,B 0,C 180,E1 -6434.871,E2 -6434.871} C_VEL
LIN {X 0,Y 488.115,Z 441.926,A -85,B 0,C 180,E1 -6437.412,E2 -6437.412} C_VEL
LIN {X 0,Y 488.005,Z 445.103,A -85,B 0,C 180,E1 -6440.679,E2 -6440.679} C_VEL
LIN {X 0,Y 487.978,Z 448.178,A -85,B 0,C 180,E1 -6443.808,E2 -6443.808} C_VEL
LIN {X 0,Y 488,Z 448.736,A -85,B 0,C 180,E1 -6444.32,E2 -6444.32} C_VEL
LIN {X 0,Y 491.679,Z 463.207,A -85,B 0,C 180,E1 -6444.827,E2 -6444.827} C_VEL
LIN {X 0,Y 492.153,Z 466.983,A -85,B 0,C 180,E1 -6444.971,E2 -6444.971} C_VEL
LIN {X 0,Y 491.773,Z 481.119,A -85,B 0,C 180,E1 -6445.545,E2 -6445.545} C_VEL
LIN {X 0,Y 491.282,Z 493.615,A -85,B 0,C 180,E1 -6446.212,E2 -6446.212} C_VEL
LIN {X 0,Y 490.77,Z 505.828,A -85,B 0,C 180,E1 -6447.031,E2 -6447.031} C_VEL
LIN {X 0,Y 490.231,Z 517.156,A -85,B 0,C 180,E1 -6447.965,E2 -6447.965} C_VEL
LIN {X 0,Y 489.71,Z 528.266,A -85,B 0,C 180,E1 -6449.077,E2 -6449.077} C_VEL
LIN {X 0,Y 489.283,Z 538.279,A -85,B 0,C 180,E1 -6450.293,E2 -6450.293} C_VEL
LIN {X 0,Y 488.789,Z 547.609,A -85,B 0,C 180,E1 -6451.674,E2 -6451.674} C_VEL
LIN {X 0,Y 488.492,Z 555.55,A -85,B 0,C 180,E1 -6453.124,E2 -6453.124} C_VEL
LIN {X 0,Y 488.264,Z 561.357,A -85,B 0,C 180,E1 -6454.417,E2 -6454.417} C_VEL
LIN {X 0,Y 488.115,Z 566.277,A -85,B 0,C 180,E1 -6455.773,E2 -6455.773} C_VEL
LIN {X 0,Y 488.002,Z 570.205,A -85,B 0,C 180,E1 -6457.174,E2 -6457.174} C_VEL
LIN {X 0,Y 487.873,Z 573.633,A -85,B 0,C 180,E1 -6458.891,E2 -6458.891} C_VEL
LIN {X 0,Y 487.829,Z 575.562,A -85,B 0,C 180,E1 -6460.649,E2 -6460.649} C_VEL
LIN {X 0,Y 487.829,Z 576.015,A -85,B 0,C 180,E1 -6462.39,E2 -6462.39} C_VEL
LIN {X 0,Y 487.829,Z 575.04,A -85,B 0,C 180,E1 -6464.114,E2 -6464.114} C_VEL
LIN {X 0,Y 487.887,Z 572.648,A -85,B 0,C 180,E1 -6465.825,E2 -6465.825} C_VEL
LIN {X 0,Y 488.062,Z 568.791,A -85,B 0,C 180,E1 -6467.526,E2 -6467.526} C_VEL
LIN {X 0,Y 488.16,Z 564.846,A -85,B 0,C 180,E1 -6468.793,E2 -6468.793} C_VEL
LIN {X 0,Y 488.351,Z 559.968,A -85,B 0,C 180,E1 -6470.055,E2 -6470.055} C_VEL
LIN {X 0,Y 488.624,Z 552.961,A -85,B 0,C 180,E1 -6471.522,E2 -6471.522} C_VEL
LIN {X 0,Y 488.99,Z 544.999,A -85,B 0,C 180,E1 -6472.874,E2 -6472.874} C_VEL
LIN {X 0,Y 489.433,Z 535.259,A -85,B 0,C 180,E1 -6474.231,E2 -6474.231} C_VEL
LIN {X 0,Y 489.836,Z 526.273,A -85,B 0,C 180,E1 -6475.268,E2 -6475.268} C_VEL
LIN {X 0,Y 490.402,Z 514.423,A -85,B 0,C 180,E1 -6476.405,E2 -6476.405} C_VEL
LIN {X 0,Y 490.955,Z 502.47,A -85,B 0,C 180,E1 -6477.333,E2 -6477.333} C_VEL
LIN {X 0,Y 491.527,Z 489.158,A -85,B 0,C 180,E1 -6478.156,E2 -6478.156} C_VEL
LIN {X 0,Y 492.01,Z 475.42,A -85,B 0,C 180,E1 -6478.813,E2 -6478.813} C_VEL
LIN {X 0,Y 492.088,Z 465.335,A -85,B 0,C 180,E1 -6479.195,E2 -6479.195} C_VEL
LIN {X 0,Y 489.952,Z 456.347,A -85,B 0,C 180,E1 -6479.536,E2 -6479.536} C_VEL
LIN {X 0,Y 488.107,Z 449.843,A -85,B 0,C 180,E1 -6479.773,E2 -6479.773} C_VEL
LIN {X 0,Y 488.205,Z 446.729,A -85,B 0,C 180,E1 -6483.301,E2 -6483.301} C_VEL
LIN {X 0,Y 488.305,Z 445.29,A -85,B 0,C 180,E1 -6484.954,E2 -6484.954} C_VEL
LIN {X 0,Y 488.378,Z 443.191,A -85,B 0,C 180,E1 -6487.441,E2 -6487.441} C_VEL
LIN {X 0,Y 488.451,Z 440.412,A -85,B 0,C 180,E1 -6490.78,E2 -6490.78} C_VEL
LIN {X 0,Y 488.48,Z 438.375,A -85,B 0,C 180,E1 -6493.309,E2 -6493.309} C_VEL
LIN {X 0,Y 488.543,Z 436.35,A -85,B 0,C 180,E1 -6495.862,E2 -6495.862} C_VEL
LIN {X 0,Y 488.683,Z 434.363,A -85,B 0,C 180,E1 -6498.445,E2 -6498.445} C_VEL
LIN {X 0,Y 488.639,Z 433.247,A -85,B 0,C 180,E1 -6500.193,E2 -6500.193} C_VEL
LIN {X 0,Y 488.703,Z 433.236,A -85,B 0,C 180,E1 -6503.021,E2 -6503.021} C_VEL
LIN {X 0,Y 488.745,Z 433.231,A -85,B 0,C 180,E1 -6505.556,E2 -6505.556} C_VEL
LIN {X 0,Y 488.741,Z 433.233,A -85,B 0,C 180,E1 -6508.329,E2 -6508.329} C_VEL
LIN {X 0,Y 488.691,Z 433.236,A -85,B 0,C 180,E1 -6511.18,E2 -6511.18} C_VEL
LIN {X 0,Y 488.73,Z 433.235,A -85,B 0,C 180,E1 -6514.113,E2 -6514.113} C_VEL
LIN {X 0,Y 488.678,Z 433.238,A -85,B 0,C 180,E1 -6517.159,E2 -6517.159} C_VEL
LIN {X 0,Y 488.738,Z 433.232,A -85,B 0,C 180,E1 -6519.251,E2 -6519.251} C_VEL
LIN {X 0,Y 488.727,Z 433.236,A -85,B 0,C 180,E1 -6522.522,E2 -6522.522} C_VEL
LIN {X 0,Y 488.724,Z 433.243,A -85,B 0,C 180,E1 -6525.005,E2 -6525.005} C_VEL
LIN {X 0,Y 489.335,Z 436.84,A -85,B 0,C 180,E1 -6527.544,E2 -6527.544} C_VEL
LIN {X 0,Y 490.055,Z 440.635,A -85,B 0,C 180,E1 -6529.808,E2 -6529.808} C_VEL
LIN {X 0,Y 490.293,Z 443.713,A -85,B 0,C 180,E1 -6531.426,E2 -6531.426} C_VEL
LIN {X 0,Y 490.051,Z 447.927,A -85,B 0,C 180,E1 -6533.429,E2 -6533.429} C_VEL
LIN {X 0,Y 489.593,Z 454.741,A -85,B 0,C 180,E1 -6536.364,E2 -6536.364} C_VEL
LIN {X 0,Y 489.295,Z 461.003,A -85,B 0,C 180,E1 -6538.864,E2 -6538.864} C_VEL
LIN {X 0,Y 489.022,Z 468.505,A -85,B 0,C 180,E1 -6541.689,E2 -6541.689} C_VEL
LIN {X 0,Y 488.803,Z 476.222,A -85,B 0,C 180,E1 -6544.448,E2 -6544.448} C_VEL
LIN {X 0,Y 488.608,Z 485.379,A -85,B 0,C 180,E1 -6547.594,E2 -6547.594} C_VEL
LIN {X 0,Y 488.414,Z 494.617,A -85,B 0,C 180,E1 -6550.674,E2 -6550.674} C_VEL
LIN {X 0,Y 488.352,Z 499.325,A -85,B 0,C 180,E1 -6552.213,E2 -6552.213} C_VEL
LIN {X 0,Y 491.025,Z 514.667,A -85,B 0,C 180,E1 -6552.658,E2 -6552.658} C_VEL
LIN {X 0,Y 491.951,Z 521.171,A -85,B 0,C 180,E1 -6552.891,E2 -6552.891} C_VEL
LIN {X 0,Y 491.577,Z 533.962,A -85,B 0,C 180,E1 -6553.385,E2 -6553.385} C_VEL
LIN {X 0,Y 491.067,Z 546.458,A -85,B 0,C 180,E1 -6554.013,E2 -6554.013} C_VEL
LIN {X 0,Y 490.566,Z 559.463,A -85,B 0,C 180,E1 -6554.844,E2 -6554.844} C_VEL
LIN {X 0,Y 489.994,Z 571.375,A -85,B 0,C 180,E1 -6555.782,E2 -6555.782} C_VEL
LIN {X 0,Y 489.437,Z 583.296,A -85,B 0,C 180,E1 -6556.929,E2 -6556.929} C_VEL
LIN {X 0,Y 489.104,Z 593.062,A -85,B 0,C 180,E1 -6558.069,E2 -6558.069} C_VEL
LIN {X 0,Y 488.631,Z 602.79,A -85,B 0,C 180,E1 -6559.433,E2 -6559.433} C_VEL
LIN {X 0,Y 488.346,Z 611.249,A -85,B 0,C 180,E1 -6560.892,E2 -6560.892} C_VEL
LIN {X 0,Y 488.151,Z 617.146,A -85,B 0,C 180,E1 -6562.139,E2 -6562.139} C_VEL
LIN {X 0,Y 488.091,Z 622.318,A -85,B 0,C 180,E1 -6563.478,E2 -6563.478} C_VEL
LIN {X 0,Y 487.962,Z 627.011,A -85,B 0,C 180,E1 -6565.043,E2 -6565.043} C_VEL
LIN {X 0,Y 487.956,Z 630.51,A -85,B 0,C 180,E1 -6566.697,E2 -6566.697} C_VEL
LIN {X 0,Y 487.888,Z 632.582,A -85,B 0,C 180,E1 -6568.349,E2 -6568.349} C_VEL
LIN {X 0,Y 487.817,Z 633.276,A -85,B 0,C 180,E1 -6570,E2 -6570} C_VEL
LIN {X 0,Y 487.888,Z 632.615,A -85,B 0,C 180,E1 -6571.651,E2 -6571.651} C_VEL
LIN {X 0,Y 487.956,Z 630.583,A -85,B 0,C 180,E1 -6573.303,E2 -6573.303} C_VEL
LIN {X 0,Y 487.962,Z 627.128,A -85,B 0,C 180,E1 -6574.957,E2 -6574.957} C_VEL
LIN {X 0,Y 488.047,Z 622.637,A -85,B 0,C 180,E1 -6576.477,E2 -6576.477} C_VEL
LIN {X 0,Y 488.151,Z 617.353,A -85,B 0,C 180,E1 -6577.861,E2 -6577.861} C_VEL
LIN {X 0,Y 488.406,Z 610.397,A -85,B 0,C 180,E1 -6579.316,E2 -6579.316} C_VEL
LIN {X 0,Y 488.726,Z 601.764,A -85,B 0,C 180,E1 -6580.774,E2 -6580.774} C_VEL
LIN {X 0,Y 489.14,Z 591.708,A -85,B 0,C 180,E1 -6582.159,E2 -6582.159} C_VEL
LIN {X 0,Y 489.637,Z 580.879,A -85,B 0,C 180,E1 -6583.382,E2 -6583.382} C_VEL
LIN {X 0,Y 490.128,Z 569.645,A -85,B 0,C 180,E1 -6584.426,E2 -6584.426} C_VEL
LIN {X 0,Y 490.76,Z 557.269,A -85,B 0,C 180,E1 -6585.363,E2 -6585.363} C_VEL
LIN {X 0,Y 491.219,Z 545.412,A -85,B 0,C 180,E1 -6586.093,E2 -6586.093} C_VEL
LIN {X 0,Y 491.735,Z 531.777,A -85,B 0,C 180,E1 -6586.748,E2 -6586.748} C_VEL
LIN {X 0,Y 491.95,Z 519.309,A -85,B 0,C 180,E1 -6587.206,E2 -6587.206} C_VEL
LIN {X 0,Y 489.369,Z 505.735,A -85,B 0,C 180,E1 -6587.65,E2 -6587.65} C_VEL
LIN {X 0,Y 488.367,Z 500.231,A -85,B 0,C 180,E1 -6587.812,E2 -6587.812} C_VEL
LIN {X 0,Y 488.572,Z 491.47,A -85,B 0,C 180,E1 -6590.77,E2 -6590.77} C_VEL
LIN {X 0,Y 488.805,Z 482.902,A -85,B 0,C 180,E1 -6593.739,E2 -6593.739} C_VEL
LIN {X 0,Y 489.112,Z 473.678,A -85,B 0,C 180,E1 -6597.017,E2 -6597.017} C_VEL
LIN {X 0,Y 489.422,Z 465.101,A -85,B 0,C 180,E1 -6600.171,E2 -6600.171} C_VEL
LIN {X 0,Y 489.724,Z 458.783,A -85,B 0,C 180,E1 -6602.557,E2 -6602.557} C_VEL
LIN {X 0,Y 490.078,Z 451.19,A -85,B 0,C 180,E1 -6605.538,E2 -6605.538} C_VEL
LIN {X 0,Y 490.359,Z 445.043,A -85,B 0,C 180,E1 -6608.045,E2 -6608.045} C_VEL
LIN {X 0,Y 490.159,Z 441.213,A -85,B 0,C 180,E1 -6609.687,E2 -6609.687} C_VEL
LIN {X 0,Y 489.07,Z 435.109,A -85,B 0,C 180,E1 -6612.484,E2 -6612.484} C_VEL
LIN {X 0,Y 488.694,Z 433.24,A -85,B 0,C 180,E1 -6613.429,E2 -6613.429} C_VEL
LIN {X 0,Y 488.713,Z 433.236,A -85,B 0,C 180,E1 -6616.349,E2 -6616.349} C_VEL
LIN {X 0,Y 488.714,Z 433.233,A -85,B 0,C 180,E1 -6618.585,E2 -6618.585} C_VEL
LIN {X 0,Y 488.676,Z 433.242,A -85,B 0,C 180,E1 -6621.8,E2 -6621.8} C_VEL
LIN {X 0,Y 488.722,Z 433.234,A -85,B 0,C 180,E1 -6625.051,E2 -6625.051} C_VEL
LIN {X 0,Y 488.701,Z 433.234,A -85,B 0,C 180,E1 -6628.045,E2 -6628.045} C_VEL
LIN {X 0,Y 488.728,Z 433.233,A -85,B 0,C 180,E1 -6630.73,E2 -6630.73} C_VEL
LIN {X 0,Y 488.76,Z 433.228,A -85,B 0,C 180,E1 -6633.528,E2 -6633.528} C_VEL
LIN {X 0,Y 488.687,Z 433.237,A -85,B 0,C 180,E1 -6636.254,E2 -6636.254} C_VEL
LIN {X 0,Y 488.739,Z 433.231,A -85,B 0,C 180,E1 -6639.175,E2 -6639.175} C_VEL
LIN {X 0,Y 488.752,Z 433.228,A -85,B 0,C 180,E1 -6641.627,E2 -6641.627} C_VEL
LIN {X 0,Y 488.755,Z 433.231,A -85,B 0,C 180,E1 -6645,E2 -6645} C_VEL
LIN {X 0,Y 488.801,Z 433.224,A -85,B 0,C 180,E1 -6648.388,E2 -6648.388} C_VEL
LIN {X 0,Y 488.812,Z 433.222,A -85,B 0,C 180,E1 -6651.734,E2 -6651.734} C_VEL
LIN {X 0,Y 488.85,Z 433.217,A -85,B 0,C 180,E1 -6654.224,E2 -6654.224} C_VEL
LIN {X 0,Y 488.955,Z 433.205,A -85,B 0,C 180,E1 -6657.529,E2 -6657.529} C_VEL
LIN {X 0,Y 488.962,Z 433.202,A -85,B 0,C 180,E1 -6660,E2 -6660} C_VEL
LIN {X 0,Y 488.957,Z 433.204,A -85,B 0,C 180,E1 -6662.472,E2 -6662.472} C_VEL
LIN {X 0,Y 488.867,Z 433.216,A -85,B 0,C 180,E1 -6665.776,E2 -6665.776} C_VEL
LIN {X 0,Y 488.812,Z 433.223,A -85,B 0,C 180,E1 -6668.267,E2 -6668.267} C_VEL
LIN {X 0,Y 488.799,Z 433.225,A -85,B 0,C 180,E1 -6671.613,E2 -6671.613} C_VEL
LIN {X 0,Y 488.756,Z 433.229,A -85,B 0,C 180,E1 -6675.001,E2 -6675.001} C_VEL
LIN {X 0,Y 488.749,Z 433.231,A -85,B 0,C 180,E1 -6678.443,E2 -6678.443} C_VEL
LIN {X 0,Y 488.702,Z 433.236,A -85,B 0,C 180,E1 -6681.071,E2 -6681.071} C_VEL
LIN {X 0,Y 488.689,Z 433.239,A -85,B 0,C 180,E1 -6683.746,E2 -6683.746} C_VEL
LIN {X 0,Y 488.787,Z 433.224,A -85,B 0,C 180,E1 -6686.944,E2 -6686.944} C_VEL
LIN {X 0,Y 488.706,Z 433.237,A -85,B 0,C 180,E1 -6690.364,E2 -6690.364} C_VEL
LIN {X 0,Y 488.732,Z 433.234,A -85,B 0,C 180,E1 -6693.485,E2 -6693.485} C_VEL
LIN {X 0,Y 488.685,Z 433.239,A -85,B 0,C 180,E1 -6696.356,E2 -6696.356} C_VEL
LIN {X 0,Y 488.698,Z 433.236,A -85,B 0,C 180,E1 -6699.255,E2 -6699.255} C_VEL
LIN {X 0,Y 488.721,Z 433.235,A -85,B 0,C 180,E1 -6701.603,E2 -6701.603} C_VEL
LIN {X 0,Y 488.71,Z 433.233,A -85,B 0,C 180,E1 -6704.802,E2 -6704.802} C_VEL
LIN {X 0,Y 488.69,Z 433.238,A -85,B 0,C 180,E1 -6707.475,E2 -6707.475} C_VEL
LIN {X 0,Y 488.732,Z 433.233,A -85,B 0,C 180,E1 -6709.677,E2 -6709.677} C_VEL
LIN {X 0,Y 488.68,Z 433.24,A -85,B 0,C 180,E1 -6712.278,E2 -6712.278} C_VEL
LIN {X 0,Y 488.729,Z 433.232,A -85,B 0,C 180,E1 -6715.052,E2 -6715.052} C_VEL
LIN {X 0,Y 488.706,Z 433.238,A -85,B 0,C 180,E1 -6718.046,E2 -6718.046} C_VEL
LIN {X 0,Y 488.733,Z 433.233,A -85,B 0,C 180,E1 -6720.766,E2 -6720.766} C_VEL
LIN {X 0,Y 488.759,Z 433.231,A -85,B 0,C 180,E1 -6723.529,E2 -6723.529} C_VEL
LIN {X 0,Y 488.745,Z 433.23,A -85,B 0,C 180,E1 -6724.357,E2 -6724.357} C_VEL
LIN {X 0,Y 488.101,Z 433.313,A -85,B 0,C 180,E1 -6725.045,E2 -6725.045} C_VEL
LIN {X 0,Y 485.232,Z 433.674,A -85,B 0,C 180,E1 -6726.161,E2 -6726.161} C_VEL
LIN {X 0,Y 482.785,Z 433.978,A -85,B 0,C 180,E1 -6727.061,E2 -6727.061} C_VEL
LIN {X 0,Y 481.727,Z 434.107,A -85,B 0,C 180,E1 -6727.757,E2 -6727.757} C_VEL
LIN {X 0,Y 481.638,Z 434.116,A -85,B 0,C 180,E1 -6727.992,E2 -6727.992} C_VEL
LIN {X 0,Y 481.708,Z 434.108,A -85,B 0,C 180,E1 -6730.394,E2 -6730.394} C_VEL
LIN {X 0,Y 481.692,Z 434.109,A -85,B 0,C 180,E1 -6733.034,E2 -6733.034} C_VEL
LIN {X 0,Y 481.694,Z 434.11,A -85,B 0,C 180,E1 -6735.639,E2 -6735.639} C_VEL
LIN {X 0,Y 481.755,Z 434.101,A -85,B 0,C 180,E1 -6738.215,E2 -6738.215} C_VEL
LIN {X 0,Y 481.766,Z 434.101,A -85,B 0,C 180,E1 -6741.612,E2 -6741.612} C_VEL
LIN {X 0,Y 481.781,Z 434.097,A -85,B 0,C 180,E1 -6744.979,E2 -6744.979} C_VEL
LIN {X 0,Y 481.932,Z 434.079,A -85,B 0,C 180,E1 -6747.493,E2 -6747.493} C_VEL
LIN {X 0,Y 481.89,Z 434.084,A -85,B 0,C 180,E1 -6750.836,E2 -6750.836} C_VEL
LIN {X 0,Y 481.932,Z 434.08,A -85,B 0,C 180,E1 -6752.507,E2 -6752.507} C_VEL
LIN {X 0,Y 481.821,Z 434.092,A -85,B 0,C 180,E1 -6755.86,E2 -6755.86} C_VEL
LIN {X 0,Y 481.745,Z 434.102,A -85,B 0,C 180,E1 -6758.388,E2 -6758.388} C_VEL
LIN {X 0,Y 481.755,Z 434.103,A -85,B 0,C 180,E1 -6761.785,E2 -6761.785} C_VEL
LIN {X 0,Y 481.746,Z 434.103,A -85,B 0,C 180,E1 -6765.224,E2 -6765.224} C_VEL
LIN {X 0,Y 481.715,Z 434.106,A -85,B 0,C 180,E1 -6768.721,E2 -6768.721} C_VEL
LIN {X 0,Y 481.649,Z 434.116,A -85,B 0,C 180,E1 -6771.394,E2 -6771.394} C_VEL
LIN {X 0,Y 481.68,Z 434.11,A -85,B 0,C 180,E1 -6774.113,E2 -6774.113} C_VEL
LIN {X 0,Y 481.749,Z 434.105,A -85,B 0,C 180,E1 -6777.139,E2 -6777.139} C_VEL
LIN {X 0,Y 481.681,Z 434.112,A -85,B 0,C 180,E1 -6779.74,E2 -6779.74} C_VEL
LIN {X 0,Y 481.651,Z 434.116,A -85,B 0,C 180,E1 -6782.675,E2 -6782.675} C_VEL
LIN {X 0,Y 481.538,Z 434.132,A -85,B 0,C 180,E1 -6785.183,E2 -6785.183} C_VEL
LIN {X 0,Y 481.211,Z 434.172,A -85,B 0,C 180,E1 -6787.939,E2 -6787.939} C_VEL
LIN {X 0,Y 481.112,Z 434.848,A -85,B 0,C 180,E1 -6789.266,E2 -6789.266} C_VEL
LIN {X 0,Y 481.059,Z 437.617,A -85,B 0,C 180,E1 -6792.223,E2 -6792.223} C_VEL
LIN {X 0,Y 481.013,Z 440.697,A -85,B 0,C 180,E1 -6795.467,E2 -6795.467} C_VEL
LIN {X 0,Y 480.99,Z 443.302,A -85,B 0,C 180,E1 -6798.174,E2 -6798.174} C_VEL
LIN {X 0,Y 480.924,Z 446.098,A -85,B 0,C 180,E1 -6801.069,E2 -6801.069} C_VEL
LIN {X 0,Y 480.911,Z 449,A -85,B 0,C 180,E1 -6804.034,E2 -6804.034} C_VEL
LIN {X 0,Y 485.084,Z 465.364,A -85,B 0,C 180,E1 -6804.649,E2 -6804.649} C_VEL
LIN {X 0,Y 485.364,Z 468.556,A -85,B 0,C 180,E1 -6804.776,E2 -6804.776} C_VEL
LIN {X 0,Y 484.922,Z 482.497,A -85,B 0,C 180,E1 -6805.364,E2 -6805.364} C_VEL
LIN {X 0,Y 484.396,Z 495.245,A -85,B 0,C 180,E1 -6806.068,E2 -6806.068} C_VEL
LIN {X 0,Y 483.799,Z 508.438,A -85,B 0,C 180,E1 -6806.993,E2 -6806.993} C_VEL
LIN {X 0,Y 483.178,Z 520.56,A -85,B 0,C 180,E1 -6808.056,E2 -6808.056} C_VEL
LIN {X 0,Y 482.654,Z 531.372,A -85,B 0,C 180,E1 -6809.215,E2 -6809.215} C_VEL
LIN {X 0,Y 482.132,Z 541.309,A -85,B 0,C 180,E1 -6810.505,E2 -6810.505} C_VEL
LIN {X 0,Y 481.71,Z 550.315,A -85,B 0,C 180,E1 -6811.932,E2 -6811.932} C_VEL
LIN {X 0,Y 481.354,Z 558.555,A -85,B 0,C 180,E1 -6813.556,E2 -6813.556} C_VEL
LIN {X 0,Y 481.138,Z 564.132,A -85,B 0,C 180,E1 -6814.937,E2 -6814.937} C_VEL
LIN {X 0,Y 480.999,Z 568.513,A -85,B 0,C 180,E1 -6816.308,E2 -6816.308} C_VEL
LIN {X 0,Y 480.876,Z 571.851,A -85,B 0,C 180,E1 -6817.667,E2 -6817.667} C_VEL
LIN {X 0,Y 480.809,Z 574.864,A -85,B 0,C 180,E1 -6819.463,E2 -6819.463} C_VEL
LIN {X 0,Y 480.767,Z 576.324,A -85,B 0,C 180,E1 -6821.24,E2 -6821.24} C_VEL
LIN {X 0,Y 480.784,Z 576.48,A -85,B 0,C 180,E1 -6822.123,E2 -6822.123} C_VEL
LIN {X 0,Y 480.73,Z 575.714,A -85,B 0,C 180,E1 -6823.873,E2 -6823.873} C_VEL
LIN {X 0,Y 480.807,Z 573.523,A -85,B 0,C 180,E1 -6825.612,E2 -6825.612} C_VEL
LIN {X 0,Y 480.993,Z 569.878,A -85,B 0,C 180,E1 -6827.339,E2 -6827.339} C_VEL
LIN {X 0,Y 481.154,Z 564.718,A -85,B 0,C 180,E1 -6829.054,E2 -6829.054} C_VEL
LIN {X 0,Y 481.355,Z 559.692,A -85,B 0,C 180,E1 -6830.334,E2 -6830.334} C_VEL
LIN {X 0,Y 481.669,Z 552.518,A -85,B 0,C 180,E1 -6831.821,E2 -6831.821} C_VEL
LIN {X 0,Y 482.034,Z 545.126,A -85,B 0,C 180,E1 -6833.073,E2 -6833.073} C_VEL
LIN {X 0,Y 482.469,Z 536.021,A -85,B 0,C 180,E1 -6834.357,E2 -6834.357} C_VEL
LIN {X 0,Y 483.016,Z 525.168,A -85,B 0,C 180,E1 -6835.619,E2 -6835.619} C_VEL
LIN {X 0,Y 483.574,Z 514.141,A -85,B 0,C 180,E1 -6836.667,E2 -6836.667} C_VEL
LIN {X 0,Y 484.158,Z 502.022,A -85,B 0,C 180,E1 -6837.608,E2 -6837.608} C_VEL
LIN {X 0,Y 484.707,Z 490.429,A -85,B 0,C 180,E1 -6838.338,E2 -6838.338} C_VEL
LIN {X 0,Y 485.177,Z 477.964,A -85,B 0,C 180,E1 -6838.962,E2 -6838.962} C_VEL
LIN {X 0,Y 485.332,Z 466.801,A -85,B 0,C 180,E1 -6839.404,E2 -6839.404} C_VEL
LIN {X 0,Y 483.46,Z 458.724,A -85,B 0,C 180,E1 -6839.728,E2 -6839.728} C_VEL
LIN {X 0,Y 481.051,Z 450.377,A -85,B 0,C 180,E1 -6840.026,E2 -6840.026} C_VEL
LIN {X 0,Y 481.298,Z 446.734,A -85,B 0,C 180,E1 -6844.187,E2 -6844.187} C_VEL
LIN {X 0,Y 481.378,Z 444.458,A -85,B 0,C 180,E1 -6846.897,E2 -6846.897} C_VEL
LIN {X 0,Y 481.353,Z 441.845,A -85,B 0,C 180,E1 -6850.091,E2 -6850.091} C_VEL
LIN {X 0,Y 481.45,Z 439.796,A -85,B 0,C 180,E1 -6852.648,E2 -6852.648} C_VEL
LIN {X 0,Y 481.529,Z 437.529,A -85,B 0,C 180,E1 -6855.578,E2 -6855.578} C_VEL
LIN {X 0,Y 481.659,Z 435.16,A -85,B 0,C 180,E1 -6858.724,E2 -6858.724} C_VEL
LIN {X 0,Y 481.601,Z 434.124,A -85,B 0,C 180,E1 -6860.501,E2 -6860.501} C_VEL
LIN {X 0,Y 481.659,Z 434.113,A -85,B 0,C 180,E1 -6863.201,E2 -6863.201} C_VEL
LIN {X 0,Y 481.7,Z 434.11,A -85,B 0,C 180,E1 -6865.957,E2 -6865.957} C_VEL
LIN {X 0,Y 481.701,Z 434.108,A -85,B 0,C 180,E1 -6868.781,E2 -6868.781} C_VEL
LIN {X 0,Y 481.655,Z 434.116,A -85,B 0,C 180,E1 -6872.19,E2 -6872.19} C_VEL
LIN {X 0,Y 481.688,Z 434.109,A -85,B 0,C 180,E1 -6874.682,E2 -6874.682} C_VEL
LIN {X 0,Y 481.653,Z 434.116,A -85,B 0,C 180,E1 -6878.008,E2 -6878.008} C_VEL
LIN {X 0,Y 481.681,Z 434.111,A -85,B 0,C 180,E1 -6880.651,E2 -6880.651} C_VEL
LIN {X 0,Y 481.68,Z 434.114,A -85,B 0,C 180,E1 -6883.295,E2 -6883.295} C_VEL
LIN {X 0,Y 481.678,Z 434.155,A -85,B 0,C 180,E1 -6884.455,E2 -6884.455} C_VEL
LIN {X 0,Y 482.209,Z 437.223,A -85,B 0,C 180,E1 -6886.78,E2 -6886.78} C_VEL
LIN {X 0,Y 482.906,Z 440.998,A -85,B 0,C 180,E1 -6889.182,E2 -6889.182} C_VEL
LIN {X 0,Y 483.32,Z 444.8,A -85,B 0,C 180,E1 -6891.299,E2 -6891.299} C_VEL
LIN {X 0,Y 483.067,Z 449.142,A -85,B 0,C 180,E1 -6893.381,E2 -6893.381} C_VEL
LIN {X 0,Y 482.573,Z 455.985,A -85,B 0,C 180,E1 -6896.399,E2 -6896.399} C_VEL
LIN {X 0,Y 482.273,Z 462.005,A -85,B 0,C 180,E1 -6898.848,E2 -6898.848} C_VEL
LIN {X 0,Y 482.045,Z 468.215,A -85,B 0,C 180,E1 -6901.242,E2 -6901.242} C_VEL
LIN {X 0,Y 481.804,Z 475.874,A -85,B 0,C 180,E1 -6904.049,E2 -6904.049} C_VEL
LIN {X 0,Y 481.545,Z 485.025,A -85,B 0,C 180,E1 -6907.274,E2 -6907.274} C_VEL
LIN {X 0,Y 481.346,Z 494.139,A -85,B 0,C 180,E1 -6910.378,E2 -6910.378} C_VEL
LIN {X 0,Y 481.29,Z 498.807,A -85,B 0,C 180,E1 -6911.936,E2 -6911.936} C_VEL
LIN {X 0,Y 484.096,Z 515.317,A -85,B 0,C 180,E1 -6912.44,E2 -6912.44} C_VEL
LIN {X 0,Y 485.121,Z 521.475,A -85,B 0,C 180,E1 -6912.677,E2 -6912.677} C_VEL
LIN {X 0,Y 484.663,Z 535.151,A -85,B 0,C 180,E1 -6913.232,E2 -6913.232} C_VEL
LIN {X 0,Y 484.066,Z 549.245,A -85,B 0,C 180,E1 -6913.987,E2 -6913.987} C_VEL
LIN {X 0,Y 483.474,Z 561.684,A -85,B 0,C 180,E1 -6914.832,E2 -6914.832} C_VEL
LIN {X 0,Y 482.836,Z 574.306,A -85,B 0,C 180,E1 -6915.889,E2 -6915.889} C_VEL
LIN {X 0,Y 482.362,Z 584.681,A -85,B 0,C 180,E1 -6916.948,E2 -6916.948} C_VEL
LIN {X 0,Y 481.972,Z 595.007,A -85,B 0,C 180,E1 -6918.221,E2 -6918.221} C_VEL
LIN {X 0,Y 481.544,Z 603.579,A -85,B 0,C 180,E1 -6919.489,E2 -6919.489} C_VEL
LIN {X 0,Y 481.241,Z 611.773,A -85,B 0,C 180,E1 -6920.968,E2 -6920.968} C_VEL
LIN {X 0,Y 481.008,Z 618.377,A -85,B 0,C 180,E1 -6922.444,E2 -6922.444} C_VEL
LIN {X 0,Y 481,Z 622.253,A -85,B 0,C 180,E1 -6923.496,E2 -6923.496} C_VEL
LIN {X 0,Y 480.896,Z 626.564,A -85,B 0,C 180,E1 -6924.97,E2 -6924.97} C_VEL
LIN {X 0,Y 480.881,Z 630.077,A -85,B 0,C 180,E1 -6926.649,E2 -6926.649} C_VEL
LIN {X 0,Y 480.819,Z 632.161,A -85,B 0,C 180,E1 -6928.325,E2 -6928.325} C_VEL
LIN {X 0,Y 480.741,Z 632.862,A -85,B 0,C 180,E1 -6930,E2 -6930} C_VEL
LIN {X 0,Y 480.819,Z 632.205,A -85,B 0,C 180,E1 -6931.675,E2 -6931.675} C_VEL
LIN {X 0,Y 480.88,Z 630.173,A -85,B 0,C 180,E1 -6933.351,E2 -6933.351} C_VEL
LIN {X 0,Y 480.896,Z 626.715,A -85,B 0,C 180,E1 -6935.03,E2 -6935.03} C_VEL
LIN {X 0,Y 480.961,Z 621.736,A -85,B 0,C 180,E1 -6936.713,E2 -6936.713} C_VEL
LIN {X 0,Y 481.147,Z 615.093,A -85,B 0,C 180,E1 -6938.399,E2 -6938.399} C_VEL
LIN {X 0,Y 481.395,Z 607.698,A -85,B 0,C 180,E1 -6939.877,E2 -6939.877} C_VEL
LIN {X 0,Y 481.821,Z 598.52,A -85,B 0,C 180,E1 -6941.356,E2 -6941.356} C_VEL
LIN {X 0,Y 482.225,Z 588.908,A -85,B 0,C 180,E1 -6942.627,E2 -6942.627} C_VEL
LIN {X 0,Y 482.78,Z 578.281,A -85,B 0,C 180,E1 -6943.79,E2 -6943.79} C_VEL
LIN {X 0,Y 483.34,Z 566.568,A -85,B 0,C 180,E1 -6944.849,E2 -6944.849} C_VEL
LIN {X 0,Y 484.01,Z 553.605,A -85,B 0,C 180,E1 -6945.798,E2 -6945.798} C_VEL
LIN {X 0,Y 484.606,Z 539.812,A -85,B 0,C 180,E1 -6946.597,E2 -6946.597} C_VEL
LIN {X 0,Y 485.099,Z 525.437,A -85,B 0,C 180,E1 -6947.222,E2 -6947.222} C_VEL
LIN {X 0,Y 485.089,Z 520.111,A -85,B 0,C 180,E1 -6947.416,E2 -6947.416} C_VEL
LIN {X 0,Y 482.427,Z 505.959,A -85,B 0,C 180,E1 -6947.897,E2 -6947.897} C_VEL
LIN {X 0,Y 481.332,Z 499.938,A -85,B 0,C 180,E1 -6948.067,E2 -6948.067} C_VEL
LIN {X 0,Y 481.512,Z 491.686,A -85,B 0,C 180,E1 -6950.913,E2 -6950.913} C_VEL
LIN {X 0,Y 481.788,Z 482.623,A -85,B 0,C 180,E1 -6954.107,E2 -6954.107} C_VEL
LIN {X 0,Y 482.076,Z 474.066,A -85,B 0,C 180,E1 -6957.215,E2 -6957.215} C_VEL
LIN {X 0,Y 482.395,Z 466.139,A -85,B 0,C 180,E1 -6960.174,E2 -6960.174} C_VEL
LIN {X 0,Y 482.737,Z 459.856,A -85,B 0,C 180,E1 -6962.593,E2 -6962.593} C_VEL
LIN {X 0,Y 483.191,Z 451.079,A -85,B 0,C 180,E1 -6966.09,E2 -6966.09} C_VEL
LIN {X 0,Y 483.408,Z 444.876,A -85,B 0,C 180,E1 -6968.693,E2 -6968.693} C_VEL
LIN {X 0,Y 482.769,Z 439.893,A -85,B 0,C 180,E1 -6970.926,E2 -6970.926} C_VEL
LIN {X 0,Y 481.648,Z 434.117,A -85,B 0,C 180,E1 -6973.726,E2 -6973.726} C_VEL
LIN {X 0,Y 481.685,Z 434.109,A -85,B 0,C 180,E1 -6976.845,E2 -6976.845} C_VEL
LIN {X 0,Y 481.672,Z 434.111,A -85,B 0,C 180,E1 -6980.059,E2 -6980.059} C_VEL
LIN {X 0,Y 481.624,Z 434.12,A -85,B 0,C 180,E1 -6983.253,E2 -6983.253} C_VEL
LIN {X 0,Y 481.704,Z 434.109,A -85,B 0,C 180,E1 -6986.33,E2 -6986.33} C_VEL
LIN {X 0,Y 481.659,Z 434.113,A -85,B 0,C 180,E1 -6989.414,E2 -6989.414} C_VEL
LIN {X 0,Y 481.697,Z 434.107,A -85,B 0,C 180,E1 -6992.168,E2 -6992.168} C_VEL
LIN {X 0,Y 481.712,Z 434.107,A -85,B 0,C 180,E1 -6994.97,E2 -6994.97} C_VEL
LIN {X 0,Y 481.646,Z 434.113,A -85,B 0,C 180,E1 -6997.705,E2 -6997.705} C_VEL
LIN {X 0,Y 481.702,Z 434.108,A -85,B 0,C 180,E1 -7000.393,E2 -7000.393} C_VEL
LIN {X 0,Y 481.686,Z 434.11,A -85,B 0,C 180,E1 -7003.034,E2 -7003.034} C_VEL
LIN {X 0,Y 481.683,Z 434.109,A -85,B 0,C 180,E1 -7005.639,E2 -7005.639} C_VEL
LIN {X 0,Y 481.746,Z 434.104,A -85,B 0,C 180,E1 -7008.215,E2 -7008.215} C_VEL
LIN {X 0,Y 481.757,Z 434.1,A -85,B 0,C 180,E1 -7011.612,E2 -7011.612} C_VEL
LIN {X 0,Y 481.811,Z 434.094,A -85,B 0,C 180,E1 -7014.14,E2 -7014.14} C_VEL
LIN {X 0,Y 481.922,Z 434.081,A -85,B 0,C 180,E1 -7017.493,E2 -7017.493} C_VEL
LIN {X 0,Y 481.933,Z 434.078,A -85,B 0,C 180,E1 -7020,E2 -7020} C_VEL
LIN {X 0,Y 481.923,Z 434.08,A -85,B 0,C 180,E1 -7022.508,E2 -7022.508} C_VEL
LIN {X 0,Y 481.825,Z 434.093,A -85,B 0,C 180,E1 -7025.86,E2 -7025.86} C_VEL
LIN {X 0,Y 481.757,Z 434.102,A -85,B 0,C 180,E1 -7028.389,E2 -7028.389} C_VEL
LIN {X 0,Y 481.744,Z 434.103,A -85,B 0,C 180,E1 -7031.785,E2 -7031.785} C_VEL
LIN {X 0,Y 481.736,Z 434.104,A -85,B 0,C 180,E1 -7035.225,E2 -7035.225} C_VEL
LIN {X 0,Y 481.707,Z 434.107,A -85,B 0,C 180,E1 -7038.722,E2 -7038.722} C_VEL
LIN {X 0,Y 481.641,Z 434.115,A -85,B 0,C 180,E1 -7041.395,E2 -7041.395} C_VEL
LIN {X 0,Y 481.672,Z 434.113,A -85,B 0,C 180,E1 -7044.114,E2 -7044.114} C_VEL
LIN {X 0,Y 481.742,Z 434.101,A -85,B 0,C 180,E1 -7047.14,E2 -7047.14} C_VEL
LIN {X 0,Y 481.674,Z 434.112,A -85,B 0,C 180,E1 -7049.742,E2 -7049.742} C_VEL
LIN {X 0,Y 481.669,Z 434.112,A -85,B 0,C 180,E1 -7052.675,E2 -7052.675} C_VEL
LIN {X 0,Y 481.639,Z 434.115,A -85,B 0,C 180,E1 -7055.71,E2 -7055.71} C_VEL
LIN {X 0,Y 481.667,Z 434.113,A -85,B 0,C 180,E1 -7058.86,E2 -7058.86} C_VEL
LIN {X 0,Y 481.66,Z 434.114,A -85,B 0,C 180,E1 -7061.915,E2 -7061.915} C_VEL
LIN {X 0,Y 481.658,Z 434.114,A -85,B 0,C 180,E1 -7064.458,E2 -7064.458} C_VEL
LIN {X 0,Y 481.647,Z 434.115,A -85,B 0,C 180,E1 -7067.84,E2 -7067.84} C_VEL
LIN {X 0,Y 481.712,Z 434.106,A -85,B 0,C 180,E1 -7070.647,E2 -7070.647} C_VEL
LIN {X 0,Y 481.644,Z 434.115,A -85,B 0,C 180,E1 -7074.292,E2 -7074.292} C_VEL
LIN {X 0,Y 481.673,Z 434.111,A -85,B 0,C 180,E1 -7077.327,E2 -7077.327} C_VEL
LIN {X 0,Y 481.689,Z 434.11,A -85,B 0,C 180,E1 -7080.26,E2 -7080.26} C_VEL
LIN {X 0,Y 481.748,Z 434.101,A -85,B 0,C 180,E1 -7083.113,E2 -7083.113} C_VEL
LIN {X 0,Y 481.677,Z 434.112,A -85,B 0,C 180,E1 -7085.887,E2 -7085.887} C_VEL
LIN {X 0,Y 481.638,Z 434.116,A -85,B 0,C 180,E1 -7087.992,E2 -7087.992} C_VEL
LIN {X 0,Y 480.971,Z 434.198,A -85,B 0,C 180,E1 -7088.69,E2 -7088.69} C_VEL
LIN {X 0,Y 478.145,Z 434.551,A -85,B 0,C 180,E1 -7089.825,E2 -7089.825} C_VEL
LIN {X 0,Y 475.76,Z 434.848,A -85,B 0,C 180,E1 -7090.739,E2 -7090.739} C_VEL
LIN {X 0,Y 474.739,Z 434.976,A -85,B 0,C 180,E1 -7091.445,E2 -7091.445} C_VEL
LIN {X 0,Y 474.657,Z 434.986,A -85,B 0,C 180,E1 -7091.684,E2 -7091.684} C_VEL
LIN {X 0,Y 474.704,Z 434.98,A -85,B 0,C 180,E1 -7094.545,E2 -7094.545} C_VEL
LIN {X 0,Y 474.708,Z 434.979,A -85,B 0,C 180,E1 -7098.038,E2 -7098.038} C_VEL
LIN {X 0,Y 474.731,Z 434.979,A -85,B 0,C 180,E1 -7101.487,E2 -7101.487} C_VEL
LIN {X 0,Y 474.751,Z 434.973,A -85,B 0,C 180,E1 -7104.904,E2 -7104.904} C_VEL
LIN {X 0,Y 474.898,Z 434.956,A -85,B 0,C 180,E1 -7107.455,E2 -7107.455} C_VEL
LIN {X 0,Y 474.916,Z 434.952,A -85,B 0,C 180,E1 -7110,E2 -7110} C_VEL
LIN {X 0,Y 474.898,Z 434.956,A -85,B 0,C 180,E1 -7112.545,E2 -7112.545} C_VEL
LIN {X 0,Y 474.783,Z 434.969,A -85,B 0,C 180,E1 -7115.947,E2 -7115.947} C_VEL
LIN {X 0,Y 474.717,Z 434.977,A -85,B 0,C 180,E1 -7118.514,E2 -7118.514} C_VEL
LIN {X 0,Y 474.708,Z 434.98,A -85,B 0,C 180,E1 -7121.962,E2 -7121.962} C_VEL
LIN {X 0,Y 474.703,Z 434.98,A -85,B 0,C 180,E1 -7125.455,E2 -7125.455} C_VEL
LIN {X 0,Y 474.668,Z 434.987,A -85,B 0,C 180,E1 -7129.01,E2 -7129.01} C_VEL
LIN {X 0,Y 474.592,Z 434.994,A -85,B 0,C 180,E1 -7131.728,E2 -7131.728} C_VEL
LIN {X 0,Y 474.662,Z 434.986,A -85,B 0,C 180,E1 -7134.492,E2 -7134.492} C_VEL
LIN {X 0,Y 474.701,Z 434.981,A -85,B 0,C 180,E1 -7137.338,E2 -7137.338} C_VEL
LIN {X 0,Y 474.606,Z 434.992,A -85,B 0,C 180,E1 -7140.81,E2 -7140.81} C_VEL
LIN {X 0,Y 474.614,Z 434.991,A -85,B 0,C 180,E1 -7143.222,E2 -7143.222} C_VEL
LIN {X 0,Y 474.493,Z 435.009,A -85,B 0,C 180,E1 -7145.448,E2 -7145.448} C_VEL
LIN {X 0,Y 474.091,Z 435.06,A -85,B 0,C 180,E1 -7148.506,E2 -7148.506} C_VEL
LIN {X 0,Y 474.02,Z 437.013,A -85,B 0,C 180,E1 -7150.874,E2 -7150.874} C_VEL
LIN {X 0,Y 473.995,Z 440.11,A -85,B 0,C 180,E1 -7154.176,E2 -7154.176} C_VEL
LIN {X 0,Y 473.929,Z 442.783,A -85,B 0,C 180,E1 -7156.988,E2 -7156.988} C_VEL
LIN {X 0,Y 473.885,Z 446.134,A -85,B 0,C 180,E1 -7160.46,E2 -7160.46} C_VEL
LIN {X 0,Y 473.846,Z 449.364,A -85,B 0,C 180,E1 -7163.784,E2 -7163.784} C_VEL
LIN {X 0,Y 477.82,Z 464.263,A -85,B 0,C 180,E1 -7164.336,E2 -7164.336} C_VEL
LIN {X 0,Y 478.578,Z 469.496,A -85,B 0,C 180,E1 -7164.553,E2 -7164.553} C_VEL
LIN {X 0,Y 478.08,Z 483.735,A -85,B 0,C 180,E1 -7165.17,E2 -7165.17} C_VEL
LIN {X 0,Y 477.523,Z 496.618,A -85,B 0,C 180,E1 -7165.905,E2 -7165.905} C_VEL
LIN {X 0,Y 476.893,Z 509.408,A -85,B 0,C 180,E1 -7166.831,E2 -7166.831} C_VEL
LIN {X 0,Y 476.24,Z 521.425,A -85,B 0,C 180,E1 -7167.909,E2 -7167.909} C_VEL
LIN {X 0,Y 475.666,Z 532.733,A -85,B 0,C 180,E1 -7169.154,E2 -7169.154} C_VEL
LIN {X 0,Y 475.082,Z 543.019,A -85,B 0,C 180,E1 -7170.536,E2 -7170.536} C_VEL
LIN {X 0,Y 474.678,Z 551.662,A -85,B 0,C 180,E1 -7171.96,E2 -7171.96} C_VEL
LIN {X 0,Y 474.392,Z 557.66,A -85,B 0,C 180,E1 -7173.16,E2 -7173.16} C_VEL
LIN {X 0,Y 474.107,Z 564.077,A -85,B 0,C 180,E1 -7174.719,E2 -7174.719} C_VEL
LIN {X 0,Y 473.927,Z 569.394,A -85,B 0,C 180,E1 -7176.397,E2 -7176.397} C_VEL
LIN {X 0,Y 473.842,Z 571.645,A -85,B 0,C 180,E1 -7177.317,E2 -7177.317} C_VEL
LIN {X 0,Y 473.716,Z 574.89,A -85,B 0,C 180,E1 -7179.141,E2 -7179.141} C_VEL
LIN {X 0,Y 473.66,Z 576.583,A -85,B 0,C 180,E1 -7180.948,E2 -7180.948} C_VEL
LIN {X 0,Y 473.704,Z 576.87,A -85,B 0,C 180,E1 -7181.846,E2 -7181.846} C_VEL
LIN {X 0,Y 473.635,Z 576.369,A -85,B 0,C 180,E1 -7183.624,E2 -7183.624} C_VEL
LIN {X 0,Y 473.738,Z 574.398,A -85,B 0,C 180,E1 -7185.392,E2 -7185.392} C_VEL
LIN {X 0,Y 473.881,Z 570.967,A -85,B 0,C 180,E1 -7187.146,E2 -7187.146} C_VEL
LIN {X 0,Y 474.061,Z 566.021,A -85,B 0,C 180,E1 -7188.888,E2 -7188.888} C_VEL
LIN {X 0,Y 474.28,Z 561.221,A -85,B 0,C 180,E1 -7190.188,E2 -7190.188} C_VEL
LIN {X 0,Y 474.584,Z 554.303,A -85,B 0,C 180,E1 -7191.698,E2 -7191.698} C_VEL
LIN {X 0,Y 475.048,Z 545.737,A -85,B 0,C 180,E1 -7193.203,E2 -7193.203} C_VEL
LIN {X 0,Y 475.506,Z 536.815,A -85,B 0,C 180,E1 -7194.487,E2 -7194.487} C_VEL
LIN {X 0,Y 476.085,Z 526.047,A -85,B 0,C 180,E1 -7195.767,E2 -7195.767} C_VEL
LIN {X 0,Y 476.686,Z 515.122,A -85,B 0,C 180,E1 -7196.83,E2 -7196.83} C_VEL
LIN {X 0,Y 477.302,Z 503.135,A -85,B 0,C 180,E1 -7197.785,E2 -7197.785} C_VEL
LIN {X 0,Y 477.905,Z 490.422,A -85,B 0,C 180,E1 -7198.597,E2 -7198.597} C_VEL
LIN {X 0,Y 478.421,Z 477.85,A -85,B 0,C 180,E1 -7199.229,E2 -7199.229} C_VEL
LIN {X 0,Y 478.537,Z 467.606,A -85,B 0,C 180,E1 -7199.642,E2 -7199.642} C_VEL
LIN {X 0,Y 475.315,Z 455.449,A -85,B 0,C 180,E1 -7200.145,E2 -7200.145} C_VEL
LIN {X 0,Y 474.005,Z 450.898,A -85,B 0,C 180,E1 -7200.318,E2 -7200.318} C_VEL
LIN {X 0,Y 474.259,Z 447.501,A -85,B 0,C 180,E1 -7204.249,E2 -7204.249} C_VEL
LIN {X 0,Y 474.349,Z 445.247,A -85,B 0,C 180,E1 -7206.946,E2 -7206.946} C_VEL
LIN {X 0,Y 474.316,Z 442.622,A -85,B 0,C 180,E1 -7210.242,E2 -7210.242} C_VEL
LIN {X 0,Y 474.398,Z 440.574,A -85,B 0,C 180,E1 -7212.839,E2 -7212.839} C_VEL
LIN {X 0,Y 474.505,Z 437.921,A -85,B 0,C 180,E1 -7216.344,E2 -7216.344} C_VEL
LIN {X 0,Y 474.636,Z 435.991,A -85,B 0,C 180,E1 -7219.011,E2 -7219.011} C_VEL
LIN {X 0,Y 474.589,Z 434.997,A -85,B 0,C 180,E1 -7221.105,E2 -7221.105} C_VEL
LIN {X 0,Y 474.653,Z 434.988,A -85,B 0,C 180,E1 -7224.493,E2 -7224.493} C_VEL
LIN {X 0,Y 474.693,Z 434.981,A -85,B 0,C 180,E1 -7227.339,E2 -7227.339} C_VEL
LIN {X 0,Y 474.605,Z 434.992,A -85,B 0,C 180,E1 -7230.812,E2 -7230.812} C_VEL
LIN {X 0,Y 474.633,Z 434.99,A -85,B 0,C 180,E1 -7233.984,E2 -7233.984} C_VEL
LIN {X 0,Y 474.571,Z 434.996,A -85,B 0,C 180,E1 -7236.9,E2 -7236.9} C_VEL
LIN {X 0,Y 474.646,Z 434.988,A -85,B 0,C 180,E1 -7239.651,E2 -7239.651} C_VEL
LIN {X 0,Y 474.648,Z 434.989,A -85,B 0,C 180,E1 -7242.931,E2 -7242.931} C_VEL
LIN {X 0,Y 474.676,Z 435.315,A -85,B 0,C 180,E1 -7244.097,E2 -7244.097} C_VEL
LIN {X 0,Y 475.364,Z 439.294,A -85,B 0,C 180,E1 -7247.151,E2 -7247.151} C_VEL
LIN {X 0,Y 476.043,Z 442.975,A -85,B 0,C 180,E1 -7249.49,E2 -7249.49} C_VEL
LIN {X 0,Y 476.353,Z 446.484,A -85,B 0,C 180,E1 -7251.439,E2 -7251.439} C_VEL
LIN {X 0,Y 476.094,Z 450.282,A -85,B 0,C 180,E1 -7253.322,E2 -7253.322} C_VEL
LIN {X 0,Y 475.585,Z 457.037,A -85,B 0,C 180,E1 -7256.348,E2 -7256.348} C_VEL
LIN {X 0,Y 475.236,Z 463.583,A -85,B 0,C 180,E1 -7259.063,E2 -7259.063} C_VEL
LIN {X 0,Y 474.942,Z 470.453,A -85,B 0,C 180,E1 -7261.737,E2 -7261.737} C_VEL
LIN {X 0,Y 474.688,Z 478.068,A -85,B 0,C 180,E1 -7264.574,E2 -7264.574} C_VEL
LIN {X 0,Y 474.441,Z 487.134,A -85,B 0,C 180,E1 -7267.807,E2 -7267.807} C_VEL
LIN {X 0,Y 474.243,Z 496.31,A -85,B 0,C 180,E1 -7270.973,E2 -7270.973} C_VEL
LIN {X 0,Y 474.219,Z 498.334,A -85,B 0,C 180,E1 -7271.665,E2 -7271.665} C_VEL
LIN {X 0,Y 476.833,Z 513.857,A -85,B 0,C 180,E1 -7272.137,E2 -7272.137} C_VEL
LIN {X 0,Y 478.235,Z 522.892,A -85,B 0,C 180,E1 -7272.495,E2 -7272.495} C_VEL
LIN {X 0,Y 477.761,Z 536.048,A -85,B 0,C 180,E1 -7273.056,E2 -7273.056} C_VEL
LIN {X 0,Y 477.172,Z 548.647,A -85,B 0,C 180,E1 -7273.75,E2 -7273.75} C_VEL
LIN {X 0,Y 476.576,Z 561.086,A -85,B 0,C 180,E1 -7274.607,E2 -7274.607} C_VEL
LIN {X 0,Y 475.905,Z 573.717,A -85,B 0,C 180,E1 -7275.679,E2 -7275.679} C_VEL
LIN {X 0,Y 475.369,Z 584.1,A -85,B 0,C 180,E1 -7276.753,E2 -7276.753} C_VEL
LIN {X 0,Y 474.962,Z 594.455,A -85,B 0,C 180,E1 -7278.044,E2 -7278.044} C_VEL
LIN {X 0,Y 474.486,Z 603.05,A -85,B 0,C 180,E1 -7279.33,E2 -7279.33} C_VEL
LIN {X 0,Y 474.177,Z 611.274,A -85,B 0,C 180,E1 -7280.832,E2 -7280.832} C_VEL
LIN {X 0,Y 473.932,Z 617.901,A -85,B 0,C 180,E1 -7282.33,E2 -7282.33} C_VEL
LIN {X 0,Y 473.918,Z 622.153,A -85,B 0,C 180,E1 -7283.505,E2 -7283.505} C_VEL
LIN {X 0,Y 473.829,Z 626.116,A -85,B 0,C 180,E1 -7284.894,E2 -7284.894} C_VEL
LIN {X 0,Y 473.807,Z 629.644,A -85,B 0,C 180,E1 -7286.599,E2 -7286.599} C_VEL
LIN {X 0,Y 473.752,Z 631.74,A -85,B 0,C 180,E1 -7288.3,E2 -7288.3} C_VEL
LIN {X 0,Y 473.668,Z 632.448,A -85,B 0,C 180,E1 -7290,E2 -7290} C_VEL
LIN {X 0,Y 473.752,Z 631.795,A -85,B 0,C 180,E1 -7291.7,E2 -7291.7} C_VEL
LIN {X 0,Y 473.806,Z 629.762,A -85,B 0,C 180,E1 -7293.401,E2 -7293.401} C_VEL
LIN {X 0,Y 473.83,Z 626.302,A -85,B 0,C 180,E1 -7295.106,E2 -7295.106} C_VEL
LIN {X 0,Y 473.891,Z 621.317,A -85,B 0,C 180,E1 -7296.814,E2 -7296.814} C_VEL
LIN {X 0,Y 474.083,Z 614.666,A -85,B 0,C 180,E1 -7298.525,E2 -7298.525} C_VEL
LIN {X 0,Y 474.337,Z 607.261,A -85,B 0,C 180,E1 -7300.026,E2 -7300.026} C_VEL
LIN {X 0,Y 474.77,Z 598.065,A -85,B 0,C 180,E1 -7301.527,E2 -7301.527} C_VEL
LIN {X 0,Y 475.239,Z 588.444,A -85,B 0,C 180,E1 -7302.816,E2 -7302.816} C_VEL
LIN {X 0,Y 475.805,Z 577.805,A -85,B 0,C 180,E1 -7303.997,E2 -7303.997} C_VEL
LIN {X 0,Y 476.401,Z 566.08,A -85,B 0,C 180,E1 -7305.07,E2 -7305.07} C_VEL
LIN {X 0,Y 477.041,Z 554.682,A -85,B 0,C 180,E1 -7305.926,E2 -7305.926} C_VEL
LIN {X 0,Y 477.649,Z 541.764,A -85,B 0,C 180,E1 -7306.709,E2 -7306.709} C_VEL
LIN {X 0,Y 478.215,Z 527.687,A -85,B 0,C 180,E1 -7307.368,E2 -7307.368} C_VEL
LIN {X 0,Y 478.198,Z 521.191,A -85,B 0,C 180,E1 -7307.617,E2 -7307.617} C_VEL
LIN {X 0,Y 475.504,Z 506.146,A -85,B 0,C 180,E1 -7308.152,E2 -7308.152} C_VEL
LIN {X 0,Y 474.283,Z 499.627,A -85,B 0,C 180,E1 -7308.337,E2 -7308.337} C_VEL
LIN {X 0,Y 474.439,Z 491.902,A -85,B 0,C 180,E1 -7311.055,E2 -7311.055} C_VEL
LIN {X 0,Y 474.728,Z 483.623,A -85,B 0,C 180,E1 -7314.023,E2 -7314.023} C_VEL
LIN {X 0,Y 475.01,Z 476.015,A -85,B 0,C 180,E1 -7316.824,E2 -7316.824} C_VEL
LIN {X 0,Y 475.36,Z 467.177,A -85,B 0,C 180,E1 -7320.177,E2 -7320.177} C_VEL
LIN {X 0,Y 475.728,Z 460.871,A -85,B 0,C 180,E1 -7322.641,E2 -7322.641} C_VEL
LIN {X 0,Y 476.209,Z 452.157,A -85,B 0,C 180,E1 -7326.18,E2 -7326.18} C_VEL
LIN {X 0,Y 476.438,Z 446.5,A -85,B 0,C 180,E1 -7328.573,E2 -7328.573} C_VEL
LIN {X 0,Y 475.96,Z 442.201,A -85,B 0,C 180,E1 -7330.518,E2 -7330.518} C_VEL
LIN {X 0,Y 474.683,Z 435.291,A -85,B 0,C 180,E1 -7333.837,E2 -7333.837} C_VEL
LIN {X 0,Y 474.621,Z 434.993,A -85,B 0,C 180,E1 -7334.102,E2 -7334.102} C_VEL
LIN {X 0,Y 474.648,Z 434.985,A -85,B 0,C 180,E1 -7337.07,E2 -7337.07} C_VEL
LIN {X 0,Y 474.64,Z 434.99,A -85,B 0,C 180,E1 -7340.454,E2 -7340.454} C_VEL
LIN {X 0,Y 474.587,Z 434.993,A -85,B 0,C 180,E1 -7343.676,E2 -7343.676} C_VEL
LIN {X 0,Y 474.638,Z 434.988,A -85,B 0,C 180,E1 -7346.78,E2 -7346.78} C_VEL
LIN {X 0,Y 474.612,Z 434.992,A -85,B 0,C 180,E1 -7349.77,E2 -7349.77} C_VEL
LIN {X 0,Y 474.709,Z 434.98,A -85,B 0,C 180,E1 -7352.681,E2 -7352.681} C_VEL
LIN {X 0,Y 474.653,Z 434.987,A -85,B 0,C 180,E1 -7355.507,E2 -7355.507} C_VEL
LIN {X 0,Y 474.664,Z 434.985,A -85,B 0,C 180,E1 -7359.185,E2 -7359.185} C_VEL
LIN {X 0,Y 474.651,Z 434.984,A -85,B 0,C 180,E1 -7361.884,E2 -7361.884} C_VEL
LIN {X 0,Y 474.693,Z 434.981,A -85,B 0,C 180,E1 -7364.544,E2 -7364.544} C_VEL
LIN {X 0,Y 474.699,Z 434.981,A -85,B 0,C 180,E1 -7368.038,E2 -7368.038} C_VEL
LIN {X 0,Y 474.723,Z 434.976,A -85,B 0,C 180,E1 -7371.487,E2 -7371.487} C_VEL
LIN {X 0,Y 474.773,Z 434.971,A -85,B 0,C 180,E1 -7374.052,E2 -7374.052} C_VEL
LIN {X 0,Y 474.889,Z 434.957,A -85,B 0,C 180,E1 -7377.456,E2 -7377.456} C_VEL
LIN {X 0,Y 474.904,Z 434.953,A -85,B 0,C 180,E1 -7380,E2 -7380} C_VEL
LIN {X 0,Y 474.89,Z 434.957,A -85,B 0,C 180,E1 -7382.545,E2 -7382.545} C_VEL
LIN {X 0,Y 474.785,Z 434.971,A -85,B 0,C 180,E1 -7385.948,E2 -7385.948} C_VEL
LIN {X 0,Y 474.722,Z 434.98,A -85,B 0,C 180,E1 -7388.514,E2 -7388.514} C_VEL
LIN {X 0,Y 474.698,Z 434.98,A -85,B 0,C 180,E1 -7391.963,E2 -7391.963} C_VEL
LIN {X 0,Y 474.694,Z 434.981,A -85,B 0,C 180,E1 -7395.456,E2 -7395.456} C_VEL
LIN {X 0,Y 474.66,Z 434.985,A -85,B 0,C 180,E1 -7399.011,E2 -7399.011} C_VEL
LIN {X 0,Y 474.585,Z 434.993,A -85,B 0,C 180,E1 -7401.729,E2 -7401.729} C_VEL
LIN {X 0,Y 474.654,Z 434.986,A -85,B 0,C 180,E1 -7404.493,E2 -7404.493} C_VEL
LIN {X 0,Y 474.676,Z 434.981,A -85,B 0,C 180,E1 -7407.335,E2 -7407.335} C_VEL
LIN {X 0,Y 474.601,Z 434.993,A -85,B 0,C 180,E1 -7410.231,E2 -7410.231} C_VEL
LIN {X 0,Y 474.639,Z 434.988,A -85,B 0,C 180,E1 -7413.221,E2 -7413.221} C_VEL
LIN {X 0,Y 474.589,Z 434.995,A -85,B 0,C 180,E1 -7416.324,E2 -7416.324} C_VEL
LIN {X 0,Y 474.624,Z 434.989,A -85,B 0,C 180,E1 -7419.648,E2 -7419.648} C_VEL
LIN {X 0,Y 474.633,Z 434.989,A -85,B 0,C 180,E1 -7422.933,E2 -7422.933} C_VEL
LIN {X 0,Y 474.608,Z 434.994,A -85,B 0,C 180,E1 -7425.896,E2 -7425.896} C_VEL
LIN {X 0,Y 474.639,Z 434.986,A -85,B 0,C 180,E1 -7429.04,E2 -7429.04} C_VEL
LIN {X 0,Y 474.616,Z 434.991,A -85,B 0,C 180,E1 -7431.704,E2 -7431.704} C_VEL
LIN {X 0,Y 474.631,Z 434.987,A -85,B 0,C 180,E1 -7434.727,E2 -7434.727} C_VEL
LIN {X 0,Y 474.637,Z 434.989,A -85,B 0,C 180,E1 -7437.789,E2 -7437.789} C_VEL
LIN {X 0,Y 474.633,Z 434.989,A -85,B 0,C 180,E1 -7440.884,E2 -7440.884} C_VEL
LIN {X 0,Y 474.663,Z 434.988,A -85,B 0,C 180,E1 -7443.629,E2 -7443.629} C_VEL
LIN {X 0,Y 474.638,Z 434.987,A -85,B 0,C 180,E1 -7446.642,E2 -7446.642} C_VEL
LIN {X 0,Y 474.658,Z 434.987,A -85,B 0,C 180,E1 -7450.09,E2 -7450.09} C_VEL
LIN {X 0,Y 474.657,Z 434.986,A -85,B 0,C 180,E1 -7451.684,E2 -7451.684} C_VEL
LIN {X 0,Y 473.994,Z 435.071,A -85,B 0,C 180,E1 -7452.393,E2 -7452.393} C_VEL
LIN {X 0,Y 471.143,Z 435.427,A -85,B 0,C 180,E1 -7453.544,E2 -7453.544} C_VEL
LIN {X 0,Y 468.728,Z 435.726,A -85,B 0,C 180,E1 -7454.472,E2 -7454.472} C_VEL
LIN {X 0,Y 467.687,Z 435.854,A -85,B 0,C 180,E1 -7455.19,E2 -7455.19} C_VEL
LIN {X 0,Y 467.6,Z 435.863,A -85,B 0,C 180,E1 -7455.432,E2 -7455.432} C_VEL
LIN {X 0,Y 467.655,Z 435.858,A -85,B 0,C 180,E1 -7458.734,E2 -7458.734} C_VEL
LIN {X 0,Y 467.684,Z 435.856,A -85,B 0,C 180,E1 -7461.357,E2 -7461.357} C_VEL
LIN {X 0,Y 467.725,Z 435.851,A -85,B 0,C 180,E1 -7463.962,E2 -7463.962} C_VEL
LIN {X 0,Y 467.863,Z 435.832,A -85,B 0,C 180,E1 -7467.417,E2 -7467.417} C_VEL
LIN {X 0,Y 467.887,Z 435.827,A -85,B 0,C 180,E1 -7470,E2 -7470} C_VEL
LIN {X 0,Y 467.863,Z 435.832,A -85,B 0,C 180,E1 -7472.583,E2 -7472.583} C_VEL
LIN {X 0,Y 467.747,Z 435.846,A -85,B 0,C 180,E1 -7476.037,E2 -7476.037} C_VEL
LIN {X 0,Y 467.675,Z 435.854,A -85,B 0,C 180,E1 -7478.643,E2 -7478.643} C_VEL
LIN {X 0,Y 467.66,Z 435.857,A -85,B 0,C 180,E1 -7482.145,E2 -7482.145} C_VEL
LIN {X 0,Y 467.642,Z 435.86,A -85,B 0,C 180,E1 -7485.695,E2 -7485.695} C_VEL
LIN {X 0,Y 467.62,Z 435.862,A -85,B 0,C 180,E1 -7488.764,E2 -7488.764} C_VEL
LIN {X 0,Y 467.583,Z 435.868,A -85,B 0,C 180,E1 -7491.268,E2 -7491.268} C_VEL
LIN {X 0,Y 467.576,Z 435.867,A -85,B 0,C 180,E1 -7493.943,E2 -7493.943} C_VEL
LIN {X 0,Y 467.618,Z 435.863,A -85,B 0,C 180,E1 -7496.8,E2 -7496.8} C_VEL
LIN {X 0,Y 467.556,Z 435.871,A -85,B 0,C 180,E1 -7499.737,E2 -7499.737} C_VEL
LIN {X 0,Y 467.573,Z 435.871,A -85,B 0,C 180,E1 -7502.758,E2 -7502.758} C_VEL
LIN {X 0,Y 467.474,Z 435.883,A -85,B 0,C 180,E1 -7504.84,E2 -7504.84} C_VEL
LIN {X 0,Y 467.085,Z 435.931,A -85,B 0,C 180,E1 -7508.09,E2 -7508.09} C_VEL
LIN {X 0,Y 466.97,Z 436.152,A -85,B 0,C 180,E1 -7509.205,E2 -7509.205} C_VEL
LIN {X 0,Y 466.928,Z 439.174,A -85,B 0,C 180,E1 -7512.478,E2 -7512.478} C_VEL
LIN {X 0,Y 466.913,Z 441.56,A -85,B 0,C 180,E1 -7515.027,E2 -7515.027} C_VEL
LIN {X 0,Y 466.857,Z 443.921,A -85,B 0,C 180,E1 -7517.53,E2 -7517.53} C_VEL
LIN {X 0,Y 466.795,Z 447.055,A -85,B 0,C 180,E1 -7520.776,E2 -7520.776} C_VEL
LIN {X 0,Y 466.804,Z 449.83,A -85,B 0,C 180,E1 -7523.51,E2 -7523.51} C_VEL
LIN {X 0,Y 470.848,Z 464.833,A -85,B 0,C 180,E1 -7524.083,E2 -7524.083} C_VEL
LIN {X 0,Y 471.792,Z 470.165,A -85,B 0,C 180,E1 -7524.316,E2 -7524.316} C_VEL
LIN {X 0,Y 471.284,Z 484.378,A -85,B 0,C 180,E1 -7524.947,E2 -7524.947} C_VEL
LIN {X 0,Y 470.685,Z 497.164,A -85,B 0,C 180,E1 -7525.69,E2 -7525.69} C_VEL
LIN {X 0,Y 470.083,Z 509.119,A -85,B 0,C 180,E1 -7526.563,E2 -7526.563} C_VEL
LIN {X 0,Y 469.423,Z 521.09,A -85,B 0,C 180,E1 -7527.64,E2 -7527.64} C_VEL
LIN {X 0,Y 468.805,Z 531.606,A -85,B 0,C 180,E1 -7528.788,E2 -7528.788} C_VEL
LIN {X 0,Y 468.275,Z 541.278,A -85,B 0,C 180,E1 -7530.064,E2 -7530.064} C_VEL
LIN {X 0,Y 467.72,Z 550.29,A -85,B 0,C 180,E1 -7531.505,E2 -7531.505} C_VEL
LIN {X 0,Y 467.41,Z 557.133,A -85,B 0,C 180,E1 -7532.836,E2 -7532.836} C_VEL
LIN {X 0,Y 467.073,Z 564.143,A -85,B 0,C 180,E1 -7534.528,E2 -7534.528} C_VEL
LIN {X 0,Y 466.905,Z 568.942,A -85,B 0,C 180,E1 -7536.02,E2 -7536.02} C_VEL
LIN {X 0,Y 466.789,Z 571.372,A -85,B 0,C 180,E1 -7536.955,E2 -7536.955} C_VEL
LIN {X 0,Y 466.721,Z 573.366,A -85,B 0,C 180,E1 -7537.885,E2 -7537.885} C_VEL
LIN {X 0,Y 466.643,Z 575.202,A -85,B 0,C 180,E1 -7539.027,E2 -7539.027} C_VEL
LIN {X 0,Y 466.585,Z 576.831,A -85,B 0,C 180,E1 -7540.647,E2 -7540.647} C_VEL
LIN {X 0,Y 466.613,Z 577.235,A -85,B 0,C 180,E1 -7541.599,E2 -7541.599} C_VEL
LIN {X 0,Y 466.545,Z 576.937,A -85,B 0,C 180,E1 -7543.368,E2 -7543.368} C_VEL
LIN {X 0,Y 466.637,Z 575.211,A -85,B 0,C 180,E1 -7545.165,E2 -7545.165} C_VEL
LIN {X 0,Y 466.77,Z 572.051,A -85,B 0,C 180,E1 -7546.947,E2 -7546.947} C_VEL
LIN {X 0,Y 466.895,Z 569.224,A -85,B 0,C 180,E1 -7548.07,E2 -7548.07} C_VEL
LIN {X 0,Y 467.099,Z 564.367,A -85,B 0,C 180,E1 -7549.598,E2 -7549.598} C_VEL
LIN {X 0,Y 467.411,Z 558.121,A -85,B 0,C 180,E1 -7551.134,E2 -7551.134} C_VEL
LIN {X 0,Y 467.814,Z 551.119,A -85,B 0,C 180,E1 -7552.526,E2 -7552.526} C_VEL
LIN {X 0,Y 468.292,Z 542.25,A -85,B 0,C 180,E1 -7553.97,E2 -7553.97} C_VEL
LIN {X 0,Y 468.829,Z 532.526,A -85,B 0,C 180,E1 -7555.271,E2 -7555.271} C_VEL
LIN {X 0,Y 469.479,Z 521.739,A -85,B 0,C 180,E1 -7556.46,E2 -7556.46} C_VEL
LIN {X 0,Y 470.157,Z 509.797,A -85,B 0,C 180,E1 -7557.537,E2 -7557.537} C_VEL
LIN {X 0,Y 470.828,Z 496.668,A -85,B 0,C 180,E1 -7558.487,E2 -7558.487} C_VEL
LIN {X 0,Y 471.443,Z 483.457,A -85,B 0,C 180,E1 -7559.24,E2 -7559.24} C_VEL
LIN {X 0,Y 471.875,Z 469.352,A -85,B 0,C 180,E1 -7559.854,E2 -7559.854} C_VEL
LIN {X 0,Y 469.141,Z 458.759,A -85,B 0,C 180,E1 -7560.323,E2 -7560.323} C_VEL
LIN {X 0,Y 466.959,Z 451.415,A -85,B 0,C 180,E1 -7560.625,E2 -7560.625} C_VEL
LIN {X 0,Y 467.221,Z 448.268,A -85,B 0,C 180,E1 -7564.313,E2 -7564.313} C_VEL
LIN {X 0,Y 467.308,Z 446.074,A -85,B 0,C 180,E1 -7566.986,E2 -7566.986} C_VEL
LIN {X 0,Y 467.277,Z 443.383,A -85,B 0,C 180,E1 -7570.398,E2 -7570.398} C_VEL
LIN {X 0,Y 467.355,Z 441.354,A -85,B 0,C 180,E1 -7573.036,E2 -7573.036} C_VEL
LIN {X 0,Y 467.456,Z 439.305,A -85,B 0,C 180,E1 -7575.805,E2 -7575.805} C_VEL
LIN {X 0,Y 467.633,Z 437.204,A -85,B 0,C 180,E1 -7578.773,E2 -7578.773} C_VEL
LIN {X 0,Y 467.542,Z 435.875,A -85,B 0,C 180,E1 -7581.258,E2 -7581.258} C_VEL
LIN {X 0,Y 467.567,Z 435.871,A -85,B 0,C 180,E1 -7583.943,E2 -7583.943} C_VEL
LIN {X 0,Y 467.622,Z 435.863,A -85,B 0,C 180,E1 -7586.8,E2 -7586.8} C_VEL
LIN {X 0,Y 467.582,Z 435.868,A -85,B 0,C 180,E1 -7589.736,E2 -7589.736} C_VEL
LIN {X 0,Y 467.579,Z 435.867,A -85,B 0,C 180,E1 -7592.759,E2 -7592.759} C_VEL
LIN {X 0,Y 467.552,Z 435.872,A -85,B 0,C 180,E1 -7595.89,E2 -7595.89} C_VEL
LIN {X 0,Y 467.611,Z 435.864,A -85,B 0,C 180,E1 -7599.142,E2 -7599.142} C_VEL
LIN {X 0,Y 467.615,Z 435.866,A -85,B 0,C 180,E1 -7602.572,E2 -7602.572} C_VEL
LIN {X 0,Y 467.71,Z 436.604,A -85,B 0,C 180,E1 -7603.842,E2 -7603.842} C_VEL
LIN {X 0,Y 468.252,Z 439.674,A -85,B 0,C 180,E1 -7606.338,E2 -7606.338} C_VEL
LIN {X 0,Y 468.878,Z 443.204,A -85,B 0,C 180,E1 -7608.738,E2 -7608.738} C_VEL
LIN {X 0,Y 469.192,Z 445.1,A -85,B 0,C 180,E1 -7609.903,E2 -7609.903} C_VEL
LIN {X 0,Y 469.347,Z 449.174,A -85,B 0,C 180,E1 -7612.126,E2 -7612.126} C_VEL
LIN {X 0,Y 468.738,Z 455.774,A -85,B 0,C 180,E1 -7615.268,E2 -7615.268} C_VEL
LIN {X 0,Y 468.365,Z 462.824,A -85,B 0,C 180,E1 -7618.32,E2 -7618.32} C_VEL
LIN {X 0,Y 467.952,Z 470.168,A -85,B 0,C 180,E1 -7621.276,E2 -7621.276} C_VEL
LIN {X 0,Y 467.638,Z 478.315,A -85,B 0,C 180,E1 -7624.385,E2 -7624.385} C_VEL
LIN {X 0,Y 467.393,Z 486.723,A -85,B 0,C 180,E1 -7627.454,E2 -7627.454} C_VEL
LIN {X 0,Y 467.185,Z 495.844,A -85,B 0,C 180,E1 -7630.674,E2 -7630.674} C_VEL
LIN {X 0,Y 467.141,Z 497.824,A -85,B 0,C 180,E1 -7631.363,E2 -7631.363} C_VEL
LIN {X 0,Y 469.817,Z 513.397,A -85,B 0,C 180,E1 -7631.86,E2 -7631.86} C_VEL
LIN {X 0,Y 471.403,Z 523.762,A -85,B 0,C 180,E1 -7632.288,E2 -7632.288} C_VEL
LIN {X 0,Y 470.869,Z 536.897,A -85,B 0,C 180,E1 -7632.874,E2 -7632.874} C_VEL
LIN {X 0,Y 470.234,Z 549.807,A -85,B 0,C 180,E1 -7633.615,E2 -7633.615} C_VEL
LIN {X 0,Y 469.601,Z 561.929,A -85,B 0,C 180,E1 -7634.484,E2 -7634.484} C_VEL
LIN {X 0,Y 468.892,Z 574.252,A -85,B 0,C 180,E1 -7635.571,E2 -7635.571} C_VEL
LIN {X 0,Y 468.288,Z 585.387,A -85,B 0,C 180,E1 -7636.77,E2 -7636.77} C_VEL
LIN {X 0,Y 467.863,Z 595.447,A -85,B 0,C 180,E1 -7638.08,E2 -7638.08} C_VEL
LIN {X 0,Y 467.4,Z 603.801,A -85,B 0,C 180,E1 -7639.386,E2 -7639.386} C_VEL
LIN {X 0,Y 467.074,Z 611.814,A -85,B 0,C 180,E1 -7640.91,E2 -7640.91} C_VEL
LIN {X 0,Y 466.854,Z 617.424,A -85,B 0,C 180,E1 -7642.213,E2 -7642.213} C_VEL
LIN {X 0,Y 466.847,Z 622.002,A -85,B 0,C 180,E1 -7643.503,E2 -7643.503} C_VEL
LIN {X 0,Y 466.762,Z 625.669,A -85,B 0,C 180,E1 -7644.817,E2 -7644.817} C_VEL
LIN {X 0,Y 466.734,Z 629.211,A -85,B 0,C 180,E1 -7646.547,E2 -7646.547} C_VEL
LIN {X 0,Y 466.687,Z 631.318,A -85,B 0,C 180,E1 -7648.274,E2 -7648.274} C_VEL
LIN {X 0,Y 466.597,Z 632.035,A -85,B 0,C 180,E1 -7650,E2 -7650} C_VEL
LIN {X 0,Y 466.687,Z 631.385,A -85,B 0,C 180,E1 -7651.726,E2 -7651.726} C_VEL
LIN {X 0,Y 466.715,Z 629.351,A -85,B 0,C 180,E1 -7653.453,E2 -7653.453} C_VEL
LIN {X 0,Y 466.762,Z 625.89,A -85,B 0,C 180,E1 -7655.183,E2 -7655.183} C_VEL
LIN {X 0,Y 466.822,Z 620.898,A -85,B 0,C 180,E1 -7656.917,E2 -7656.917} C_VEL
LIN {X 0,Y 467.004,Z 614.238,A -85,B 0,C 180,E1 -7658.655,E2 -7658.655} C_VEL
LIN {X 0,Y 467.294,Z 606.825,A -85,B 0,C 180,E1 -7660.178,E2 -7660.178} C_VEL
LIN {X 0,Y 467.748,Z 597.613,A -85,B 0,C 180,E1 -7661.703,E2 -7661.703} C_VEL
LIN {X 0,Y 468.231,Z 587.98,A -85,B 0,C 180,E1 -7663.011,E2 -7663.011} C_VEL
LIN {X 0,Y 468.867,Z 577.332,A -85,B 0,C 180,E1 -7664.208,E2 -7664.208} C_VEL
LIN {X 0,Y 469.513,Z 565.596,A -85,B 0,C 180,E1 -7665.297,E2 -7665.297} C_VEL
LIN {X 0,Y 470.235,Z 552.606,A -85,B 0,C 180,E1 -7666.274,E2 -7666.274} C_VEL
LIN {X 0,Y 470.863,Z 540.502,A -85,B 0,C 180,E1 -7666.999,E2 -7666.999} C_VEL
LIN {X 0,Y 471.405,Z 527.123,A -85,B 0,C 180,E1 -7667.627,E2 -7667.627} C_VEL
LIN {X 0,Y 471.293,Z 521.71,A -85,B 0,C 180,E1 -7667.842,E2 -7667.842} C_VEL
LIN {X 0,Y 468.645,Z 506.946,A -85,B 0,C 180,E1 -7668.39,E2 -7668.39} C_VEL
LIN {X 0,Y 467.201,Z 499.304,A -85,B 0,C 180,E1 -7668.613,E2 -7668.613} C_VEL
LIN {X 0,Y 467.415,Z 490.952,A -85,B 0,C 180,E1 -7671.615,E2 -7671.615} C_VEL
LIN {X 0,Y 467.75,Z 482.069,A -85,B 0,C 180,E1 -7674.878,E2 -7674.878} C_VEL
LIN {X 0,Y 468.044,Z 474.49,A -85,B 0,C 180,E1 -7677.741,E2 -7677.741} C_VEL
